C01852=1129.708,111.484,-56.807,-179.853,8.160,149.518
C01853=1129.704,111.733,-56.826,-179.851,8.164,149.518
C01854=1129.699,111.983,-56.846,-179.849,8.167,149.519
C01855=1129.694,112.232,-56.865,-179.847,8.171,149.519
C01856=1129.690,112.481,-56.884,-179.845,8.175,149.519
C01857=1129.684,112.730,-56.904,-179.843,8.178,149.520
C01858=1129.680,112.979,-56.923,-179.841,8.182,149.520
C01859=1129.674,113.228,-56.943,-179.839,8.185,149.520
C01860=1129.670,113.478,-56.962,-179.837,8.189,149.520
C01861=1129.665,113.727,-56.981,-179.835,8.193,149.521
C01862=1129.660,113.976,-57.001,-179.833,8.196,149.521
C01863=1129.655,114.226,-57.020,-179.831,8.200,149.521
C01864=1129.650,114.474,-57.040,-179.829,8.203,149.521
C01865=1129.646,114.724,-57.059,-179.828,8.207,149.522
C01866=1129.641,114.973,-57.078,-179.826,8.210,149.522
C01867=1129.636,115.222,-57.098,-179.823,8.214,149.522
C01868=1129.631,115.472,-57.117,-179.822,8.217,149.522
C01869=1129.627,115.721,-57.138,-179.820,8.220,149.523
C01870=1129.622,115.969,-57.156,-179.818,8.224,149.523
C01871=1129.618,116.184,-57.173,-179.816,8.228,149.523
C01872=1129.614,116.399,-57.190,-179.815,8.230,149.523
C01873=1129.610,116.614,-57.207,-179.813,8.233,149.524
C01874=1129.606,116.829,-57.224,-179.811,8.236,149.524
C01875=1129.601,117.043,-57.241,-179.810,8.239,149.524
C01876=1129.597,117.259,-57.258,-179.808,8.242,149.524
C01877=1129.593,117.474,-57.275,-179.806,8.245,149.525
C01878=1129.589,117.688,-57.292,-179.805,8.248,149.525
C01879=1129.584,117.938,-57.311,-179.803,8.252,149.525
C01880=1129.579,118.187,-57.331,-179.801,8.255,149.525
C01881=1129.574,118.435,-57.351,-179.799,8.259,149.525
C01882=1129.569,118.685,-57.371,-179.797,8.261,149.526
C01883=1129.565,118.935,-57.390,-179.796,8.265,149.526
C01884=1129.560,119.183,-57.409,-179.794,8.269,149.526
C01885=1129.556,119.432,-57.429,-179.792,8.272,149.527
C01886=1129.551,119.682,-57.449,-179.789,8.276,149.527
C01887=1129.546,119.931,-57.469,-179.787,8.279,149.527
C01888=1129.541,120.179,-57.489,-179.786,8.282,149.527
C01889=1129.536,120.429,-57.508,-179.784,8.286,149.528
C01890=1129.532,120.679,-57.528,-179.782,8.289,149.528
C01891=1129.527,120.928,-57.548,-179.780,8.293,149.528
C01892=1129.522,121.176,-57.568,-179.779,8.296,149.528
C01893=1129.517,121.425,-57.588,-179.777,8.299,149.528
C01894=1129.513,121.675,-57.608,-179.775,8.303,149.529
C01895=1129.508,121.925,-57.627,-179.773,8.306,149.529
C01896=1129.503,122.173,-57.647,-179.771,8.310,149.529
C01897=1129.498,122.422,-57.667,-179.770,8.313,149.530
C01898=1129.494,122.671,-57.687,-179.767,8.316,149.530
C01899=1129.489,122.921,-57.707,-179.766,8.320,149.530
C01900=1129.484,123.170,-57.728,-179.764,8.323,149.530
C01901=1129.478,123.419,-57.747,-179.762,8.326,149.531
C01902=1129.474,123.668,-57.768,-179.760,8.330,149.531
C01903=1129.469,123.918,-57.787,-179.759,8.334,149.531
C01904=1129.465,124.166,-57.808,-179.757,8.337,149.532
C01905=1129.460,124.416,-57.827,-179.755,8.340,149.532
C01906=1129.456,124.665,-57.848,-179.753,8.343,149.532
C01907=1129.450,124.914,-57.867,-179.751,8.347,149.532
C01908=1129.446,125.163,-57.887,-179.750,8.350,149.533
C01909=1129.441,125.412,-57.907,-179.748,8.353,149.533
C01910=1129.436,125.662,-57.928,-179.746,8.357,149.533
C01911=1129.431,125.911,-57.948,-179.744,8.360,149.533
C01912=1129.427,126.160,-57.968,-179.743,8.363,149.534
C01913=1129.422,126.409,-57.988,-179.741,8.367,149.534
C01914=1129.417,126.658,-58.008,-179.739,8.370,149.534
C01915=1129.413,126.907,-58.028,-179.737,8.373,149.534
C01916=1129.407,127.156,-58.049,-179.735,8.377,149.535
C01917=1129.403,127.406,-58.069,-179.733,8.381,149.535
C01918=1129.398,127.655,-58.089,-179.732,8.383,149.535
C01919=1129.394,127.904,-58.109,-179.730,8.387,149.536
C01920=1129.389,128.153,-58.129,-179.728,8.391,149.536
C01921=1129.384,128.402,-58.150,-179.727,8.393,149.536
C01922=1129.379,128.651,-58.170,-179.725,8.397,149.536
C01923=1129.374,128.900,-58.190,-179.723,8.400,149.537
C01924=1129.370,129.149,-58.210,-179.722,8.403,149.537
C01925=1129.364,129.398,-58.231,-179.720,8.407,149.537
C01926=1129.360,129.647,-58.251,-179.718,8.410,149.538
C01927=1129.356,129.863,-58.268,-179.717,8.412,149.538
C01928=1129.352,130.077,-58.286,-179.715,8.416,149.538
C01929=1129.348,130.292,-58.305,-179.713,8.419,149.538
C01930=1129.343,130.506,-58.321,-179.712,8.422,149.539
C01931=1129.340,130.721,-58.339,-179.711,8.424,149.539
C01932=1129.336,130.936,-58.356,-179.709,8.427,149.539
C01933=1129.331,131.151,-58.375,-179.708,8.430,149.539
C01934=1129.327,131.366,-58.392,-179.707,8.432,149.539
C01935=1129.323,131.615,-58.412,-179.704,8.436,149.540
C01936=1129.318,131.864,-58.433,-179.703,8.439,149.540
C01937=1129.313,132.113,-58.453,-179.701,8.443,149.540
C01938=1129.309,132.362,-58.474,-179.699,8.446,149.541
C01939=1129.304,132.611,-58.495,-179.698,8.449,149.541
C01940=1129.299,132.859,-58.515,-179.696,8.453,149.541
C01941=1129.294,133.108,-58.535,-179.695,8.455,149.541
C01942=1129.289,133.358,-58.556,-179.693,8.459,149.542
C01943=1129.284,133.607,-58.576,-179.692,8.462,149.542
C01944=1129.279,133.856,-58.597,-179.690,8.466,149.543
C01945=1129.275,134.105,-58.617,-179.688,8.469,149.543
C01946=1129.270,134.354,-58.637,-179.687,8.472,149.543
C01947=1129.266,134.604,-58.659,-179.685,8.476,149.543
C01948=1129.261,134.853,-58.679,-179.683,8.479,149.544
C01949=1129.256,135.103,-58.700,-179.681,8.482,149.544
C01950=1129.252,135.352,-58.720,-179.680,8.485,149.544
C01951=1129.247,135.600,-58.741,-179.678,8.489,149.545
C01952=1129.242,135.850,-58.762,-179.677,8.492,149.545
C01953=1129.238,136.099,-58.782,-179.675,8.495,149.545
C01954=1129.233,136.348,-58.803,-179.674,8.498,149.545
C01955=1129.228,136.597,-58.823,-179.672,8.502,149.546
C01956=1129.223,136.846,-58.844,-179.671,8.505,149.546
C01957=1129.219,137.094,-58.865,-179.669,8.508,149.547
C01958=1129.214,137.344,-58.886,-179.667,8.512,149.547
C01959=1129.209,137.593,-58.907,-179.666,8.515,149.547
C01960=1129.204,137.842,-58.928,-179.664,8.519,149.547
C01961=1129.200,138.091,-58.948,-179.663,8.522,149.548
C01962=1129.194,138.340,-58.969,-179.661,8.525,149.548
C01963=1129.190,138.589,-58.990,-179.660,8.528,149.549
C01964=1129.185,138.838,-59.010,-179.658,8.532,149.549
C01965=1129.181,139.087,-59.032,-179.657,8.535,149.549
C01966=1129.176,139.337,-59.053,-179.655,8.537,149.549
C01967=1129.172,139.586,-59.073,-179.654,8.541,149.550
C01968=1129.166,139.835,-59.094,-179.652,8.544,149.550
C01969=1129.162,140.084,-59.115,-179.651,8.548,149.550
C01970=1129.157,140.333,-59.136,-179.649,8.551,149.551
C01971=1129.152,140.582,-59.157,-179.647,8.555,149.551
C01972=1129.148,140.831,-59.178,-179.646,8.557,149.551
C01973=1129.143,141.081,-59.199,-179.644,8.561,149.552
C01974=1129.139,141.330,-59.219,-179.643,8.564,149.552
C01975=1129.134,141.578,-59.241,-179.641,8.568,149.552
C01976=1129.129,141.827,-59.261,-179.640,8.571,149.553
C01977=1129.124,142.076,-59.282,-179.638,8.574,149.553
C01978=1129.119,142.326,-59.303,-179.637,8.577,149.554
C01979=1129.115,142.574,-59.324,-179.635,8.581,149.554
C01980=1129.110,142.824,-59.346,-179.634,8.584,149.554
C01981=1129.105,143.073,-59.367,-179.633,8.587,149.555
C01982=1129.101,143.322,-59.388,-179.631,8.590,149.555
C01983=1129.096,143.536,-59.406,-179.630,8.594,149.555
C01984=1129.093,143.751,-59.424,-179.629,8.596,149.556
C01985=1129.088,143.966,-59.442,-179.627,8.599,149.556
C01986=1129.085,144.180,-59.460,-179.626,8.602,149.556
C01987=1129.080,144.395,-59.478,-179.625,8.605,149.556
C01988=1129.076,144.610,-59.497,-179.624,8.608,149.557
C01989=1129.072,144.824,-59.515,-179.622,8.611,149.557
C01990=1129.068,145.039,-59.533,-179.622,8.613,149.557
C01991=1129.063,145.288,-59.555,-179.619,8.617,149.558
C01992=1129.059,145.537,-59.575,-179.616,8.621,149.558
C01993=1129.054,145.786,-59.597,-179.613,8.625,149.558
C01994=1129.049,146.035,-59.618,-179.611,8.630,149.558
C01995=1129.045,146.284,-59.639,-179.607,8.633,149.558
C01996=1129.040,146.533,-59.660,-179.605,8.637,149.558
C01997=1129.036,146.782,-59.682,-179.603,8.641,149.559
C01998=1129.030,147.031,-59.703,-179.600,8.646,149.559
C01999=1129.026,147.280,-59.725,-179.597,8.649,149.559
C02000=1129.021,147.529,-59.745,-179.595,8.653,149.559
C02001=1129.017,147.778,-59.767,-179.592,8.657,149.559
C02002=1129.012,148.028,-59.788,-179.589,8.661,149.559
C02003=1129.007,148.276,-59.810,-179.587,8.665,149.560
C02004=1129.002,148.525,-59.832,-179.584,8.669,149.560
C02005=1128.998,148.775,-59.852,-179.581,8.673,149.560
C02006=1128.993,149.023,-59.874,-179.579,8.676,149.560
C02007=1128.988,149.272,-59.895,-179.576,8.680,149.560
C02008=1128.984,149.522,-59.917,-179.573,8.684,149.560
C02009=1128.979,149.770,-59.939,-179.571,8.688,149.561
C02010=1128.974,150.020,-59.960,-179.568,8.692,149.561
C02011=1128.969,150.269,-59.982,-179.565,8.696,149.561
C02012=1128.965,150.518,-60.003,-179.562,8.699,149.561
C02013=1128.960,150.766,-60.025,-179.560,8.703,149.561
C02014=1128.955,151.016,-60.046,-179.557,8.706,149.561
C02015=1128.951,151.265,-60.067,-179.554,8.711,149.561
C02016=1128.946,151.513,-60.089,-179.552,8.714,149.561
C02017=1128.942,151.763,-60.111,-179.549,8.718,149.562
C02018=1128.937,152.011,-60.133,-179.547,8.721,149.562
C02019=1128.932,152.261,-60.154,-179.544,8.725,149.562
C02020=1128.928,152.510,-60.176,-179.541,8.729,149.562
C02021=1128.923,152.759,-60.198,-179.539,8.733,149.562
C02022=1128.918,153.008,-60.220,-179.536,8.736,149.562
C02023=1128.914,153.256,-60.241,-179.534,8.740,149.563
C02024=1128.909,153.505,-60.263,-179.531,8.743,149.563
C02025=1128.904,153.754,-60.285,-179.528,8.748,149.563
C02026=1128.899,154.004,-60.306,-179.526,8.751,149.563
C02027=1128.894,154.253,-60.329,-179.523,8.755,149.563
C02028=1128.889,154.502,-60.350,-179.521,8.758,149.563
C02029=1128.885,154.751,-60.372,-179.518,8.761,149.563
C02030=1128.880,155.000,-60.394,-179.515,8.765,149.563
C02031=1128.876,155.249,-60.416,-179.513,8.768,149.563
C02032=1128.871,155.498,-60.438,-179.510,8.773,149.564
C02033=1128.866,155.747,-60.459,-179.508,8.776,149.564
C02034=1128.862,155.996,-60.482,-179.505,8.779,149.564
C02035=1128.857,156.245,-60.503,-179.502,8.783,149.564
C02036=1128.853,156.494,-60.525,-179.500,8.786,149.564
C02037=1128.847,156.743,-60.548,-179.498,8.790,149.564
C02038=1128.843,156.992,-60.570,-179.495,8.794,149.564
C02039=1128.839,157.206,-60.589,-179.493,8.796,149.564
C02040=1128.835,157.421,-60.608,-179.491,8.800,149.564
C02041=1128.831,157.636,-60.627,-179.488,8.803,149.564
C02042=1128.827,157.850,-60.646,-179.486,8.805,149.564
C02043=1128.823,158.065,-60.665,-179.484,8.808,149.565
C02044=1128.819,158.279,-60.684,-179.482,8.812,149.565
C02045=1128.815,158.494,-60.703,-179.480,8.814,149.565
C02046=1128.811,158.708,-60.722,-179.477,8.817,149.565
C02047=1128.806,158.956,-60.744,-179.475,8.820,149.565
C02048=1128.802,159.206,-60.766,-179.473,8.824,149.565
C02049=1128.797,159.455,-60.789,-179.469,8.827,149.565
C02050=1128.793,159.703,-60.811,-179.467,8.831,149.565
C02051=1128.788,159.953,-60.833,-179.465,8.834,149.565
C02052=1128.783,160.201,-60.855,-179.462,8.837,149.565
C02053=1128.778,160.451,-60.877,-179.460,8.841,149.566
C02054=1128.774,160.699,-60.900,-179.457,8.845,149.566
C02055=1128.770,160.948,-60.922,-179.454,8.848,149.566
C02056=1128.765,161.198,-60.944,-179.452,8.851,149.566
C02057=1128.760,161.446,-60.967,-179.450,8.854,149.566
C02058=1128.756,161.695,-60.989,-179.447,8.857,149.566
C02059=1128.751,161.944,-61.011,-179.445,8.860,149.566
C02060=1128.746,162.193,-61.034,-179.443,8.864,149.566
C02061=1128.742,162.442,-61.056,-179.440,8.868,149.566
C02062=1128.737,162.690,-61.078,-179.437,8.871,149.566
C02063=1128.732,162.940,-61.101,-179.435,8.874,149.566
C02064=1128.728,163.189,-61.123,-179.432,8.878,149.567
C02065=1128.723,163.438,-61.146,-179.430,8.881,149.567
C02066=1128.718,163.687,-61.168,-179.427,8.884,149.567
C02067=1128.714,163.936,-61.191,-179.425,8.887,149.567
C02068=1128.709,164.185,-61.213,-179.423,8.890,149.567
C02069=1128.705,164.434,-61.236,-179.420,8.893,149.567
C02070=1128.700,164.683,-61.259,-179.418,8.897,149.567
C02071=1128.695,164.931,-61.281,-179.415,8.900,149.567
C02072=1128.691,165.181,-61.303,-179.413,8.903,149.567
C02073=1128.686,165.430,-61.326,-179.411,8.906,149.567
C02074=1128.682,165.678,-61.348,-179.408,8.909,149.567
C02075=1128.677,165.927,-61.371,-179.406,8.912,149.567
C02076=1128.673,166.177,-61.394,-179.403,8.916,149.568
C02077=1128.668,166.426,-61.417,-179.401,8.919,149.568
C02078=1128.663,166.674,-61.439,-179.398,8.922,149.568
C02079=1128.658,166.923,-61.462,-179.396,8.925,149.568
C02080=1128.654,167.172,-61.485,-179.394,8.929,149.568
C02081=1128.649,167.421,-61.507,-179.391,8.932,149.568
C02082=1128.645,167.670,-61.530,-179.389,8.935,149.568
C02083=1128.640,167.919,-61.553,-179.387,8.937,149.568
C02084=1128.636,168.168,-61.575,-179.385,8.941,149.568
C02085=1128.630,168.416,-61.598,-179.382,8.944,149.568
C02086=1128.626,168.665,-61.622,-179.380,8.947,149.568
C02087=1128.622,168.915,-61.644,-179.377,8.950,149.568
C02088=1128.617,169.164,-61.667,-179.375,8.954,149.569
C02089=1128.612,169.412,-61.689,-179.373,8.957,149.569
C02090=1128.608,169.661,-61.713,-179.370,8.960,149.569
C02091=1128.603,169.911,-61.735,-179.368,8.962,149.569
C02092=1128.599,170.159,-61.758,-179.366,8.966,149.569
C02093=1128.594,170.408,-61.781,-179.364,8.969,149.569
C02094=1128.589,170.656,-61.804,-179.361,8.972,149.569
C02095=1128.585,170.872,-61.824,-179.359,8.974,149.569
C02096=1128.581,171.085,-61.844,-179.357,8.978,149.569
C02097=1128.577,171.300,-61.864,-179.355,8.980,149.569
C02098=1128.573,171.514,-61.883,-179.353,8.982,149.569
C02099=1128.570,171.729,-61.903,-179.351,8.985,149.569
C02100=1128.565,171.943,-61.923,-179.349,8.988,149.570
C02101=1128.562,172.158,-61.943,-179.347,8.990,149.570
C02102=1128.557,172.372,-61.963,-179.345,8.993,149.570
C02103=1128.553,172.621,-61.985,-179.343,8.996,149.570
C02104=1128.548,172.870,-62.009,-179.341,8.999,149.570
C02105=1128.544,173.119,-62.032,-179.339,9.002,149.570
C02106=1128.540,173.368,-62.055,-179.336,9.005,149.570
C02107=1128.535,173.617,-62.078,-179.334,9.008,149.570
C02108=1128.530,173.865,-62.101,-179.332,9.011,149.570
C02109=1128.525,174.114,-62.124,-179.330,9.014,149.570
C02110=1128.521,174.363,-62.147,-179.327,9.017,149.570
C02111=1128.516,174.612,-62.171,-179.325,9.020,149.570
C02112=1128.512,174.861,-62.194,-179.323,9.023,149.571
C02113=1128.507,175.110,-62.217,-179.321,9.026,149.571
C02114=1128.503,175.358,-62.240,-179.318,9.029,149.571
C02115=1128.498,175.607,-62.263,-179.317,9.032,149.571
C02116=1128.494,175.857,-62.287,-179.314,9.035,149.571
C02117=1128.488,176.105,-62.310,-179.312,9.038,149.571
C02118=1128.484,176.354,-62.333,-179.310,9.040,149.571
C02119=1128.480,176.603,-62.356,-179.308,9.044,149.571
C02120=1128.475,176.852,-62.379,-179.305,9.047,149.571
C02121=1128.470,177.101,-62.403,-179.304,9.049,149.572
C02122=1128.465,177.350,-62.426,-179.301,9.053,149.572
C02123=1128.461,177.599,-62.449,-179.299,9.056,149.572
C02124=1128.456,177.848,-62.473,-179.297,9.058,149.572
C02125=1128.452,178.096,-62.496,-179.295,9.061,149.572
C02126=1128.448,178.345,-62.520,-179.293,9.064,149.572
C02127=1128.443,178.594,-62.543,-179.291,9.067,149.572
C02128=1128.438,178.843,-62.566,-179.288,9.070,149.572
C02129=1128.434,179.092,-62.590,-179.287,9.073,149.572
C02130=1128.429,179.340,-62.614,-179.284,9.076,149.572
C02131=1128.425,179.589,-62.637,-179.281,9.080,149.572
C02132=1128.420,179.838,-62.660,-179.278,9.084,149.572
C02133=1128.415,180.088,-62.684,-179.275,9.087,149.572
C02134=1128.411,180.336,-62.707,-179.272,9.090,149.572
C02135=1128.407,180.585,-62.731,-179.269,9.093,149.572
C02136=1128.402,180.834,-62.754,-179.266,9.097,149.572
C02137=1128.397,181.083,-62.777,-179.263,9.100,149.572
C02138=1128.393,181.331,-62.801,-179.260,9.104,149.572
C02139=1128.388,181.580,-62.825,-179.257,9.107,149.572
C02140=1128.384,181.829,-62.848,-179.254,9.110,149.572
C02141=1128.379,182.078,-62.872,-179.251,9.114,149.572
C02142=1128.375,182.327,-62.896,-179.249,9.117,149.572
C02143=1128.370,182.575,-62.920,-179.246,9.119,149.572
C02144=1128.365,182.824,-62.943,-179.243,9.122,149.572
C02145=1128.361,183.073,-62.966,-179.240,9.126,149.572
C02146=1128.356,183.322,-62.990,-179.237,9.129,149.572
C02147=1128.351,183.571,-63.014,-179.234,9.132,149.572
C02148=1128.347,183.820,-63.039,-179.232,9.135,149.572
C02149=1128.342,184.069,-63.062,-179.229,9.138,149.572
C02150=1128.338,184.317,-63.086,-179.227,9.142,149.572
C02151=1128.333,184.531,-63.107,-179.224,9.144,149.572
C02152=1128.330,184.746,-63.127,-179.222,9.147,149.572
C02153=1128.326,184.960,-63.148,-179.219,9.150,149.572
C02154=1128.322,185.175,-63.168,-179.218,9.152,149.572
C02155=1128.318,185.389,-63.189,-179.216,9.154,149.572
C02156=1128.315,185.603,-63.209,-179.213,9.157,149.572
C02157=1128.311,185.817,-63.230,-179.211,9.159,149.572
C02158=1128.306,186.031,-63.250,-179.209,9.162,149.572
C02159=1128.303,186.280,-63.275,-179.206,9.165,149.572
C02160=1128.298,186.530,-63.298,-179.204,9.168,149.572
C02161=1128.293,186.778,-63.323,-179.201,9.171,149.572
C02162=1128.288,187.027,-63.347,-179.199,9.174,149.572
C02163=1128.284,187.276,-63.370,-179.197,9.176,149.572
C02164=1128.279,187.524,-63.394,-179.194,9.180,149.572
C02165=1128.275,187.772,-63.418,-179.192,9.183,149.572
C02166=1128.270,188.023,-63.442,-179.190,9.185,149.572
C02167=1128.266,188.271,-63.467,-179.187,9.188,149.572
C02168=1128.261,188.519,-63.491,-179.185,9.191,149.572
C02169=1128.257,188.768,-63.514,-179.183,9.194,149.572
C02170=1128.251,189.017,-63.539,-179.181,9.197,149.573
C02171=1128.248,189.266,-63.563,-179.179,9.199,149.573
C02172=1128.243,189.515,-63.587,-179.176,9.202,149.573
C02173=1128.238,189.764,-63.610,-179.174,9.204,149.573
C02174=1128.233,190.012,-63.635,-179.172,9.208,149.573
C02175=1128.229,190.261,-63.659,-179.170,9.210,149.573
C02176=1128.225,190.510,-63.684,-179.168,9.212,149.573
C02177=1128.220,190.759,-63.708,-179.165,9.215,149.573
C02178=1128.215,191.008,-63.732,-179.163,9.218,149.573
C02179=1128.211,191.256,-63.756,-179.161,9.221,149.573
C02180=1128.207,191.505,-63.780,-179.160,9.223,149.573
C02181=1128.202,191.754,-63.805,-179.158,9.226,149.573
C02182=1128.198,192.002,-63.829,-179.156,9.228,149.573
C02183=1128.192,192.251,-63.854,-179.154,9.232,149.573
C02184=1128.189,192.500,-63.878,-179.152,9.234,149.573
C02185=1128.184,192.749,-63.901,-179.150,9.236,149.573
C02186=1128.179,192.998,-63.926,-179.148,9.239,149.574
C02187=1128.174,193.246,-63.950,-179.146,9.241,149.574
C02188=1128.171,193.495,-63.975,-179.145,9.244,149.574
C02189=1128.166,193.744,-63.999,-179.143,9.246,149.574
C02190=1128.161,193.993,-64.023,-179.141,9.250,149.574
C02191=1128.157,194.241,-64.047,-179.139,9.252,149.574
C02192=1128.152,194.490,-64.072,-179.138,9.255,149.575
C02193=1128.148,194.739,-64.097,-179.136,9.257,149.575
C02194=1128.143,194.988,-64.121,-179.134,9.260,149.575
C02195=1128.139,195.237,-64.146,-179.133,9.263,149.575
C02196=1128.134,195.485,-64.170,-179.132,9.264,149.575
C02197=1128.129,195.734,-64.194,-179.130,9.267,149.575
C02198=1128.126,195.983,-64.219,-179.129,9.270,149.576
C02199=1128.120,196.232,-64.244,-179.127,9.272,149.576
C02200=1128.116,196.480,-64.268,-179.124,9.276,149.576
C02201=1128.112,196.730,-64.293,-179.119,9.280,149.576
C02202=1128.107,196.978,-64.317,-179.116,9.284,149.575
C02203=1128.102,197.227,-64.341,-179.112,9.287,149.575
C02204=1128.098,197.476,-64.366,-179.108,9.291,149.575
C02205=1128.093,197.724,-64.390,-179.104,9.295,149.575
C02206=1128.089,197.972,-64.415,-179.101,9.298,149.575
C02207=1128.085,198.187,-64.436,-179.097,9.302,149.575
C02208=1128.081,198.401,-64.458,-179.094,9.305,149.575
C02209=1128.077,198.616,-64.479,-179.091,9.308,149.574
C02210=1128.073,198.830,-64.500,-179.088,9.311,149.574
C02211=1128.070,199.044,-64.522,-179.085,9.314,149.574
C02212=1128.066,199.258,-64.543,-179.081,9.317,149.574
C02213=1128.062,199.472,-64.564,-179.079,9.320,149.574
C02214=1128.058,199.686,-64.586,-179.076,9.323,149.574
C02215=1128.053,199.935,-64.610,-179.072,9.327,149.574
C02216=1128.049,200.184,-64.635,-179.069,9.330,149.574
C02217=1128.045,200.432,-64.660,-179.065,9.334,149.573
C02218=1128.040,200.681,-64.685,-179.062,9.336,149.573
C02219=1128.035,200.930,-64.710,-179.058,9.340,149.573
C02220=1128.031,201.178,-64.735,-179.055,9.343,149.573
C02221=1128.026,201.427,-64.760,-179.052,9.346,149.573
C02222=1128.021,201.676,-64.784,-179.048,9.350,149.573
C02223=1128.018,201.925,-64.809,-179.045,9.352,149.573
C02224=1128.013,202.173,-64.834,-179.042,9.356,149.572
C02225=1128.008,202.422,-64.860,-179.039,9.359,149.572
C02226=1128.004,202.671,-64.884,-179.035,9.362,149.572
C02227=1128.000,202.919,-64.910,-179.032,9.365,149.572
C02228=1127.995,203.168,-64.934,-179.029,9.368,149.572
C02229=1127.990,203.417,-64.960,-179.026,9.371,149.572
C02230=1127.986,203.665,-64.984,-179.023,9.374,149.572
C02231=1127.982,203.914,-65.010,-179.020,9.377,149.571
C02232=1127.977,204.163,-65.035,-179.017,9.380,149.572
C02233=1127.973,204.412,-65.060,-179.014,9.383,149.571
C02234=1127.969,204.661,-65.085,-179.011,9.386,149.571
C02235=1127.964,204.909,-65.110,-179.008,9.389,149.571
C02236=1127.960,205.158,-65.136,-179.005,9.392,149.571
C02237=1127.955,205.406,-65.161,-179.002,9.394,149.571
C02238=1127.950,205.655,-65.186,-178.999,9.397,149.571
C02239=1127.945,205.904,-65.211,-178.996,9.400,149.571
C02240=1127.941,206.153,-65.237,-178.994,9.403,149.571
C02241=1127.937,206.401,-65.262,-178.991,9.406,149.571
C02242=1127.932,206.650,-65.287,-178.988,9.409,149.571
C02243=1127.928,206.899,-65.312,-178.986,9.411,149.570
C02244=1127.923,207.147,-65.338,-178.984,9.414,149.571
C02245=1127.919,207.396,-65.363,-178.981,9.417,149.570
C02246=1127.915,207.645,-65.388,-178.978,9.420,149.570
C02247=1127.910,207.893,-65.414,-178.976,9.422,149.570
C02248=1127.905,208.142,-65.440,-178.973,9.425,149.570
C02249=1127.901,208.390,-65.465,-178.970,9.428,149.570
C02250=1127.896,208.640,-65.490,-178.968,9.430,149.570
C02251=1127.892,208.888,-65.516,-178.966,9.433,149.570
C02252=1127.887,209.136,-65.541,-178.964,9.435,149.570
C02253=1127.884,209.385,-65.566,-178.961,9.438,149.570
C02254=1127.879,209.634,-65.592,-178.959,9.441,149.570
C02255=1127.874,209.882,-65.617,-178.957,9.444,149.570
C02256=1127.870,210.131,-65.642,-178.955,9.446,149.570
C02257=1127.866,210.380,-65.668,-178.953,9.448,149.570
C02258=1127.861,210.628,-65.694,-178.950,9.451,149.570
C02259=1127.857,210.877,-65.719,-178.948,9.454,149.570
C02260=1127.853,211.126,-65.745,-178.947,9.456,149.571
C02261=1127.848,211.374,-65.771,-178.944,9.459,149.571
C02262=1127.843,211.623,-65.796,-178.943,9.462,149.571
C02263=1127.839,211.837,-65.818,-178.941,9.464,149.571
C02264=1127.835,212.051,-65.840,-178.939,9.466,149.571
C02265=1127.831,212.265,-65.862,-178.937,9.468,149.571
C02266=1127.828,212.480,-65.885,-178.936,9.471,149.571
C02267=1127.824,212.694,-65.907,-178.935,9.472,149.571
C02268=1127.820,212.908,-65.929,-178.933,9.475,149.571
C02269=1127.816,213.121,-65.951,-178.931,9.477,149.572
C02270=1127.812,213.335,-65.973,-178.931,9.479,149.572
C02271=1127.808,213.584,-65.999,-178.929,9.482,149.572
C02272=1127.804,213.833,-66.024,-178.927,9.485,149.572
C02273=1127.799,214.081,-66.050,-178.925,9.487,149.572
C02274=1127.795,214.330,-66.076,-178.923,9.490,149.572
C02275=1127.790,214.579,-66.101,-178.921,9.492,149.572
C02276=1127.786,214.828,-66.127,-178.919,9.496,149.572
C02277=1127.781,215.076,-66.153,-178.917,9.498,149.573
C02278=1127.776,215.325,-66.179,-178.915,9.501,149.573
C02279=1127.772,215.574,-66.204,-178.913,9.504,149.573
C02280=1127.768,215.822,-66.230,-178.911,9.506,149.573
C02281=1127.763,216.070,-66.256,-178.909,9.510,149.573
C02282=1127.759,216.319,-66.282,-178.907,9.512,149.573
C02283=1127.755,216.567,-66.308,-178.905,9.515,149.573
C02284=1127.751,216.816,-66.334,-178.903,9.519,149.574
C02285=1127.745,217.065,-66.360,-178.901,9.521,149.574
C02286=1127.741,217.313,-66.385,-178.898,9.524,149.574
C02287=1127.737,217.562,-66.411,-178.896,9.528,149.574
C02288=1127.733,217.810,-66.438,-178.894,9.530,149.574
C02289=1127.729,218.059,-66.463,-178.892,9.533,149.574
C02290=1127.723,218.308,-66.489,-178.889,9.536,149.574
C02291=1127.719,218.556,-66.515,-178.887,9.540,149.574
C02292=1127.715,218.805,-66.541,-178.885,9.542,149.575
C02293=1127.711,219.053,-66.567,-178.883,9.545,149.575
C02294=1127.706,219.303,-66.594,-178.880,9.548,149.575
C02295=1127.701,219.551,-66.619,-178.878,9.551,149.575
C02296=1127.697,219.800,-66.645,-178.875,9.554,149.575
C02297=1127.693,220.048,-66.671,-178.873,9.558,149.575
C02298=1127.688,220.297,-66.698,-178.871,9.561,149.575
C02299=1127.684,220.546,-66.723,-178.868,9.564,149.575
C02300=1127.680,220.794,-66.750,-178.865,9.567,149.575
C02301=1127.675,221.043,-66.776,-178.863,9.570,149.575
C02302=1127.670,221.292,-66.802,-178.860,9.573,149.575
C02303=1127.666,221.539,-66.828,-178.858,9.577,149.575
C02304=1127.662,221.788,-66.854,-178.855,9.580,149.575
C02305=1127.657,222.036,-66.881,-178.852,9.584,149.576
C02306=1127.653,222.285,-66.907,-178.849,9.586,149.575
C02307=1127.648,222.534,-66.933,-178.847,9.589,149.575
C02308=1127.644,222.783,-66.959,-178.844,9.593,149.576
C02309=1127.640,223.031,-66.985,-178.841,9.596,149.576
C02310=1127.635,223.280,-67.012,-178.838,9.600,149.576
C02311=1127.631,223.529,-67.038,-178.835,9.603,149.576
C02312=1127.626,223.777,-67.065,-178.832,9.606,149.576
C02313=1127.621,224.025,-67.090,-178.830,9.609,149.576
C02314=1127.617,224.273,-67.117,-178.826,9.613,149.576
C02315=1127.612,224.523,-67.143,-178.824,9.616,149.576
C02316=1127.609,224.771,-67.170,-178.821,9.620,149.576
C02317=1127.604,225.020,-67.196,-178.818,9.623,149.576
C02318=1127.600,225.268,-67.222,-178.814,9.626,149.576
C02319=1127.596,225.482,-67.246,-178.812,9.629,149.576
C02320=1127.592,225.696,-67.268,-178.809,9.632,149.576
C02321=1127.588,225.910,-67.291,-178.806,9.635,149.575
C02322=1127.585,226.124,-67.314,-178.804,9.638,149.576
C02323=1127.581,226.338,-67.337,-178.801,9.641,149.575
C02324=1127.577,226.551,-67.360,-178.798,9.644,149.575
C02325=1127.573,226.766,-67.382,-178.795,9.647,149.575
C02326=1127.569,226.980,-67.405,-178.792,9.649,149.575
C02327=1127.565,227.228,-67.432,-178.790,9.653,149.575
C02328=1127.560,227.477,-67.459,-178.786,9.656,149.575
C02329=1127.556,227.725,-67.485,-178.782,9.660,149.575
C02330=1127.551,227.974,-67.511,-178.779,9.663,149.575
C02331=1127.547,228.222,-67.538,-178.775,9.667,149.575
C02332=1127.543,228.471,-67.565,-178.772,9.669,149.575
C02333=1127.538,228.719,-67.592,-178.769,9.673,149.575
C02334=1127.534,228.967,-67.619,-178.765,9.676,149.574
C02335=1127.529,229.216,-67.645,-178.762,9.680,149.574
C02336=1127.526,229.465,-67.672,-178.758,9.683,149.574
C02337=1127.521,229.714,-67.699,-178.754,9.687,149.574
C02338=1127.517,229.962,-67.726,-178.751,9.691,149.574
C02339=1127.513,230.211,-67.752,-178.747,9.694,149.574
C02340=1127.508,230.459,-67.779,-178.743,9.697,149.574
C02341=1127.503,230.708,-67.806,-178.740,9.701,149.573
C02342=1127.499,230.956,-67.833,-178.737,9.703,149.573
C02343=1127.495,231.204,-67.860,-178.733,9.707,149.573
C02344=1127.490,231.453,-67.887,-178.730,9.711,149.573
C02345=1127.486,231.702,-67.914,-178.726,9.713,149.573
C02346=1127.481,231.950,-67.941,-178.723,9.716,149.573
C02347=1127.478,232.199,-67.968,-178.719,9.720,149.573
C02348=1127.473,232.447,-67.995,-178.716,9.723,149.572
C02349=1127.468,232.696,-68.022,-178.713,9.725,149.572
C02350=1127.464,232.944,-68.049,-178.710,9.729,149.572
C02351=1127.460,233.192,-68.076,-178.707,9.732,149.572
C02352=1127.456,233.441,-68.103,-178.703,9.735,149.572
C02353=1127.451,233.690,-68.130,-178.700,9.738,149.572
C02354=1127.447,233.938,-68.158,-178.697,9.740,149.571
C02355=1127.442,234.186,-68.185,-178.694,9.743,149.571
C02356=1127.437,234.435,-68.212,-178.690,9.747,149.571
C02357=1127.434,234.684,-68.239,-178.687,9.749,149.571
C02358=1127.429,234.932,-68.266,-178.684,9.752,149.571
C02359=1127.425,235.180,-68.294,-178.681,9.755,149.571
C02360=1127.420,235.429,-68.321,-178.678,9.758,149.571
C02361=1127.416,235.678,-68.348,-178.675,9.760,149.571
C02362=1127.412,235.926,-68.375,-178.673,9.763,149.571
C02363=1127.407,236.174,-68.403,-178.670,9.766,149.571
C02364=1127.403,236.423,-68.430,-178.667,9.769,149.570
C02365=1127.398,236.672,-68.457,-178.665,9.771,149.570
C02366=1127.395,236.920,-68.484,-178.662,9.774,149.570
C02367=1127.390,237.168,-68.512,-178.659,9.776,149.570
C02368=1127.386,237.416,-68.539,-178.656,9.779,149.570
C02369=1127.382,237.666,-68.566,-178.654,9.782,149.570
C02370=1127.377,237.913,-68.594,-178.651,9.784,149.570
C02371=1127.372,238.162,-68.621,-178.648,9.787,149.570
C02372=1127.368,238.410,-68.649,-178.646,9.789,149.570
C02373=1127.364,238.659,-68.676,-178.643,9.792,149.570
C02374=1127.359,238.908,-68.703,-178.641,9.794,149.569
C02375=1127.356,239.122,-68.728,-178.639,9.796,149.569
C02376=1127.352,239.335,-68.751,-178.637,9.798,149.569
C02377=1127.348,239.549,-68.774,-178.634,9.800,149.569
C02378=1127.344,239.762,-68.799,-178.633,9.803,149.569
C02379=1127.341,239.976,-68.822,-178.630,9.805,149.569
C02380=1127.337,240.190,-68.846,-178.628,9.807,149.569
C02381=1127.333,240.404,-68.870,-178.626,9.809,149.569
C02382=1127.330,240.617,-68.894,-178.624,9.811,149.569
C02383=1127.325,240.866,-68.921,-178.622,9.814,149.569
C02384=1127.321,241.115,-68.949,-178.620,9.816,149.569
C02385=1127.317,241.363,-68.976,-178.618,9.818,149.569
C02386=1127.312,241.611,-69.004,-178.615,9.821,149.569
C02387=1127.308,241.860,-69.032,-178.613,9.823,149.569
C02388=1127.303,242.108,-69.059,-178.611,9.825,149.569
C02389=1127.299,242.357,-69.086,-178.609,9.828,149.569
C02390=1127.295,242.605,-69.115,-178.607,9.830,149.569
C02391=1127.290,242.854,-69.142,-178.606,9.832,149.569
C02392=1127.286,243.102,-69.170,-178.603,9.834,149.569
C02393=1127.282,243.350,-69.198,-178.601,9.837,149.569
C02394=1127.277,243.599,-69.225,-178.599,9.839,149.569
C02395=1127.274,243.847,-69.253,-178.598,9.841,149.569
C02396=1127.269,244.096,-69.281,-178.596,9.843,149.569
C02397=1127.264,244.344,-69.308,-178.595,9.846,149.570
C02398=1127.260,244.593,-69.336,-178.593,9.848,149.570
C02399=1127.256,244.841,-69.364,-178.591,9.850,149.570
C02400=1127.252,245.090,-69.392,-178.589,9.853,149.570
C02401=1127.247,245.338,-69.419,-178.588,9.854,149.570
C02402=1127.242,245.586,-69.448,-178.586,9.857,149.570
C02403=1127.238,245.835,-69.475,-178.585,9.859,149.570
C02404=1127.234,246.083,-69.503,-178.584,9.861,149.570
C02405=1127.230,246.331,-69.531,-178.582,9.863,149.570
C02406=1127.225,246.580,-69.558,-178.581,9.865,149.570
C02407=1127.221,246.829,-69.587,-178.579,9.868,149.571
C02408=1127.217,247.077,-69.615,-178.578,9.870,149.571
C02409=1127.212,247.325,-69.642,-178.576,9.872,149.571
C02410=1127.208,247.574,-69.670,-178.572,9.876,149.571
C02411=1127.203,247.822,-69.698,-178.565,9.881,149.570
C02412=1127.199,248.071,-69.726,-178.559,9.886,149.570
C02413=1127.195,248.318,-69.754,-178.553,9.891,149.569
C02414=1127.191,248.567,-69.782,-178.546,9.896,149.569
C02415=1127.186,248.815,-69.811,-178.540,9.900,149.568
C02416=1127.182,249.064,-69.839,-178.535,9.905,149.568
C02417=1127.178,249.312,-69.867,-178.529,9.909,149.568
C02418=1127.173,249.561,-69.895,-178.524,9.914,149.567
C02419=1127.169,249.809,-69.922,-178.519,9.917,149.567
C02420=1127.165,250.057,-69.952,-178.514,9.921,149.566
C02421=1127.160,250.305,-69.980,-178.509,9.925,149.566
C02422=1127.157,250.554,-70.008,-178.505,9.928,149.566
C02423=1127.152,250.802,-70.036,-178.500,9.932,149.565
C02424=1127.148,251.050,-70.064,-178.496,9.935,149.565
C02425=1127.143,251.299,-70.093,-178.493,9.938,149.565
C02426=1127.139,251.547,-70.121,-178.489,9.941,149.565
C02427=1127.134,251.796,-70.149,-178.486,9.943,149.564
C02428=1127.130,252.044,-70.177,-178.483,9.946,149.564
C02429=1127.126,252.292,-70.207,-178.480,9.949,149.564
C02430=1127.122,252.541,-70.235,-178.478,9.951,149.564
C02431=1127.118,252.754,-70.259,-178.475,9.953,149.564
C02432=1127.114,252.968,-70.283,-178.473,9.955,149.564
C02433=1127.111,253.181,-70.308,-178.471,9.956,149.563
C02434=1127.107,253.395,-70.332,-178.470,9.957,149.563
C02435=1127.103,253.609,-70.357,-178.469,9.959,149.564
C02436=1127.100,253.823,-70.382,-178.467,9.961,149.564
C02437=1127.097,254.037,-70.406,-178.466,9.962,149.564
C02438=1127.092,254.250,-70.430,-178.465,9.964,149.564
C02439=1127.088,254.498,-70.460,-178.464,9.964,149.564
C02440=1127.084,254.747,-70.488,-178.463,9.966,149.564
C02441=1127.079,254.995,-70.516,-178.463,9.967,149.564
C02442=1127.075,255.244,-70.544,-178.463,9.969,149.564
C02443=1127.071,255.492,-70.574,-178.463,9.969,149.565
C02444=1127.066,255.740,-70.602,-178.463,9.970,149.565
C02445=1127.062,255.989,-70.630,-178.463,9.972,149.565
C02446=1127.058,256.237,-70.659,-178.460,9.974,149.565
C02447=1127.054,256.485,-70.687,-178.458,9.977,149.565
C02448=1127.049,256.734,-70.716,-178.455,9.980,149.565
C02449=1127.046,256.982,-70.744,-178.452,9.983,149.565
C02450=1127.041,257.230,-70.773,-178.449,9.986,149.565
C02451=1127.036,257.479,-70.802,-178.446,9.988,149.565
C02452=1127.033,257.727,-70.830,-178.443,9.991,149.565
C02453=1127.028,257.975,-70.859,-178.440,9.994,149.564
C02454=1127.024,258.223,-70.887,-178.437,9.997,149.564
C02455=1127.020,258.472,-70.917,-178.434,10.000,149.564
C02456=1127.015,258.720,-70.945,-178.431,10.003,149.564
C02457=1127.011,258.968,-70.973,-178.428,10.006,149.564
C02458=1127.007,259.217,-71.003,-178.424,10.009,149.564
C02459=1127.002,259.465,-71.031,-178.421,10.012,149.564
C02460=1126.998,259.713,-71.060,-178.418,10.014,149.564
C02461=1126.994,259.962,-71.089,-178.414,10.018,149.563
C02462=1126.990,260.210,-71.118,-178.411,10.021,149.563
C02463=1126.985,260.458,-71.147,-178.409,10.024,149.563
C02464=1126.981,260.706,-71.176,-178.405,10.027,149.563
C02465=1126.977,260.955,-71.204,-178.402,10.029,149.563
C02466=1126.972,261.203,-71.234,-178.398,10.033,149.563
C02467=1126.968,261.451,-71.263,-178.395,10.035,149.562
C02468=1126.964,261.699,-71.291,-178.391,10.039,149.562
C02469=1126.960,261.948,-71.320,-178.388,10.042,149.562
C02470=1126.956,262.196,-71.350,-178.384,10.045,149.562
C02471=1126.951,262.445,-71.379,-178.381,10.048,149.562
C02472=1126.947,262.692,-71.407,-178.377,10.051,149.562
C02473=1126.943,262.940,-71.437,-178.373,10.054,149.561
C02474=1126.938,263.189,-71.465,-178.370,10.057,149.561
C02475=1126.934,263.437,-71.495,-178.366,10.060,149.561
C02476=1126.930,263.686,-71.524,-178.362,10.063,149.561
C02477=1126.925,263.934,-71.553,-178.359,10.067,149.561
C02478=1126.921,264.182,-71.582,-178.355,10.070,149.560
C02479=1126.916,264.430,-71.612,-178.351,10.073,149.560
C02480=1126.913,264.678,-71.640,-178.349,10.075,149.560
C02481=1126.909,264.927,-71.670,-178.346,10.078,149.560
C02482=1126.904,265.176,-71.699,-178.343,10.080,149.560
C02483=1126.900,265.424,-71.728,-178.341,10.082,149.560
C02484=1126.895,265.671,-71.757,-178.338,10.085,149.560
C02485=1126.891,265.920,-71.787,-178.336,10.087,149.559
C02486=1126.887,266.168,-71.816,-178.333,10.090,149.559
C02487=1126.883,266.381,-71.841,-178.331,10.091,149.559
C02488=1126.880,266.595,-71.866,-178.329,10.093,149.559
C02489=1126.876,266.808,-71.892,-178.327,10.096,149.559
C02490=1126.872,267.022,-71.917,-178.324,10.098,149.559
C02491=1126.868,267.236,-71.942,-178.322,10.100,149.559
C02492=1126.865,267.449,-71.967,-178.320,10.102,149.559
C02493=1126.862,267.664,-71.993,-178.317,10.104,149.559
C02494=1126.858,267.877,-72.018,-178.316,10.106,149.559
C02495=1126.854,268.125,-72.047,-178.313,10.109,149.559
C02496=1126.849,268.373,-72.076,-178.310,10.111,149.559
C02497=1126.845,268.621,-72.106,-178.307,10.114,149.558
C02498=1126.841,268.869,-72.135,-178.305,10.116,149.558
C02499=1126.837,269.118,-72.165,-178.302,10.118,149.558
C02500=1126.832,269.366,-72.194,-178.299,10.121,149.558
C02501=1126.828,269.614,-72.224,-178.296,10.124,149.558
C02502=1126.823,269.863,-72.254,-178.294,10.126,149.558
C02503=1126.819,270.110,-72.284,-178.291,10.129,149.558
C02504=1126.815,270.359,-72.313,-178.288,10.131,149.558
C02505=1126.811,270.607,-72.343,-178.285,10.134,149.558
C02506=1126.807,270.855,-72.372,-178.283,10.136,149.557
C02507=1126.803,271.103,-72.402,-178.280,10.139,149.557
C02508=1126.799,271.352,-72.431,-178.277,10.142,149.557
C02509=1126.794,271.600,-72.460,-178.274,10.144,149.557
C02510=1126.790,271.848,-72.490,-178.271,10.147,149.557
C02511=1126.786,272.096,-72.520,-178.268,10.150,149.557
C02512=1126.781,272.344,-72.550,-178.266,10.152,149.557
C02513=1126.777,272.593,-72.580,-178.263,10.155,149.557
C02514=1126.773,272.841,-72.609,-178.260,10.157,149.556
C02515=1126.769,273.089,-72.638,-178.257,10.160,149.556
C02516=1126.765,273.337,-72.669,-178.254,10.163,149.556
C02517=1126.761,273.585,-72.698,-178.251,10.165,149.556
C02518=1126.756,273.834,-72.728,-178.248,10.168,149.556
C02519=1126.752,274.081,-72.758,-178.245,10.171,149.556
C02520=1126.748,274.330,-72.788,-178.241,10.173,149.556
C02521=1126.744,274.578,-72.817,-178.239,10.176,149.556
C02522=1126.739,274.826,-72.847,-178.236,10.179,149.555
C02523=1126.735,275.074,-72.877,-178.233,10.181,149.555
C02524=1126.731,275.322,-72.907,-178.230,10.184,149.555
C02525=1126.727,275.571,-72.937,-178.226,10.187,149.555
C02526=1126.723,275.819,-72.967,-178.223,10.189,149.555
C02527=1126.718,276.068,-72.997,-178.220,10.193,149.555
C02528=1126.714,276.315,-73.027,-178.217,10.195,149.554
C02529=1126.710,276.564,-73.057,-178.214,10.198,149.554
C02530=1126.706,276.811,-73.087,-178.211,10.201,149.554
C02531=1126.701,277.060,-73.117,-178.207,10.203,149.554
C02532=1126.698,277.307,-73.147,-178.204,10.206,149.554
C02533=1126.693,277.556,-73.177,-178.200,10.209,149.554
C02534=1126.689,277.804,-73.208,-178.197,10.212,149.554
C02535=1126.685,278.053,-73.237,-178.195,10.215,149.553
C02536=1126.681,278.301,-73.268,-178.191,10.217,149.553
C02537=1126.676,278.549,-73.297,-178.188,10.220,149.553
C02538=1126.672,278.796,-73.327,-178.184,10.223,149.553
C02539=1126.668,279.045,-73.357,-178.181,10.226,149.553
C02540=1126.664,279.293,-73.388,-178.178,10.228,149.552
C02541=1126.660,279.541,-73.418,-178.174,10.231,149.552
C02542=1126.655,279.790,-73.448,-178.171,10.234,149.552
C02543=1126.652,280.002,-73.474,-178.168,10.237,149.552
C02544=1126.648,280.216,-73.500,-178.165,10.239,149.552
C02545=1126.645,280.430,-73.527,-178.162,10.241,149.552
C02546=1126.641,280.643,-73.553,-178.159,10.244,149.551
C02547=1126.637,280.856,-73.578,-178.156,10.247,149.551
C02548=1126.634,281.069,-73.604,-178.153,10.248,149.551
C02549=1126.630,281.284,-73.630,-178.151,10.251,149.551
C02550=1126.627,281.497,-73.656,-178.147,10.253,149.550
C02551=1126.622,281.744,-73.687,-178.144,10.256,149.550
C02552=1126.619,281.993,-73.718,-178.141,10.259,149.550
C02553=1126.614,282.241,-73.748,-178.138,10.261,149.550
C02554=1126.610,282.489,-73.778,-178.135,10.264,149.550
C02555=1126.605,282.737,-73.809,-178.132,10.266,149.550
C02556=1126.601,282.985,-73.839,-178.129,10.268,149.550
C02557=1126.598,283.233,-73.870,-178.126,10.271,149.549
C02558=1126.593,283.481,-73.901,-178.123,10.274,149.549
C02559=1126.589,283.730,-73.930,-178.120,10.276,149.549
C02560=1126.585,283.978,-73.961,-178.117,10.279,149.549
C02561=1126.581,284.226,-73.991,-178.114,10.282,149.549
C02562=1126.576,284.474,-74.022,-178.111,10.284,149.548
C02563=1126.572,284.722,-74.053,-178.108,10.287,149.548
C02564=1126.568,284.970,-74.083,-178.104,10.289,149.548
C02565=1126.564,285.218,-74.114,-178.102,10.291,149.548
C02566=1126.560,285.466,-74.144,-178.099,10.294,149.548
C02567=1126.556,285.714,-74.176,-178.096,10.296,149.548
C02568=1126.551,285.962,-74.206,-178.093,10.299,149.547
C02569=1126.547,286.210,-74.236,-178.089,10.302,149.547
C02570=1126.543,286.458,-74.267,-178.086,10.304,149.547
C02571=1126.539,286.707,-74.298,-178.083,10.307,149.547
C02572=1126.535,286.954,-74.329,-178.080,10.310,149.547
C02573=1126.530,287.202,-74.359,-178.077,10.312,149.546
C02574=1126.526,287.451,-74.390,-178.074,10.315,149.546
C02575=1126.522,287.699,-74.421,-178.071,10.316,149.546
C02576=1126.518,287.947,-74.452,-178.068,10.319,149.546
C02577=1126.514,288.195,-74.482,-178.065,10.322,149.546
C02578=1126.509,288.443,-74.513,-178.062,10.324,149.546
C02579=1126.506,288.691,-74.544,-178.059,10.327,149.545
C02580=1126.502,288.939,-74.575,-178.056,10.329,149.545
C02581=1126.497,289.187,-74.606,-178.053,10.332,149.545
C02582=1126.493,289.435,-74.637,-178.049,10.335,149.545
C02583=1126.488,289.683,-74.668,-178.046,10.337,149.545
C02584=1126.485,289.932,-74.698,-178.043,10.340,149.544
C02585=1126.481,290.179,-74.730,-178.040,10.343,149.544
C02586=1126.476,290.427,-74.761,-178.038,10.344,149.544
C02587=1126.472,290.676,-74.792,-178.035,10.347,149.544
C02588=1126.468,290.924,-74.823,-178.032,10.350,149.544
C02589=1126.465,291.171,-74.854,-178.028,10.352,149.544
C02590=1126.460,291.419,-74.885,-178.025,10.355,149.544
C02591=1126.456,291.668,-74.916,-178.022,10.357,149.543
C02592=1126.452,291.915,-74.947,-178.019,10.360,149.543
C02593=1126.448,292.164,-74.978,-178.016,10.363,149.543
C02594=1126.443,292.412,-75.009,-178.013,10.365,149.543
C02595=1126.439,292.659,-75.040,-178.009,10.368,149.543
C02596=1126.435,292.908,-75.071,-178.007,10.371,149.542
C02597=1126.431,293.156,-75.102,-178.004,10.372,149.542
C02598=1126.427,293.404,-75.134,-178.001,10.375,149.542
C02599=1126.423,293.617,-75.160,-177.998,10.378,149.542
C02600=1126.420,293.831,-75.187,-177.995,10.379,149.542
C02601=1126.416,294.043,-75.214,-177.993,10.381,149.542
C02602=1126.413,294.257,-75.241,-177.990,10.384,149.541
C02603=1126.409,294.470,-75.268,-177.988,10.386,149.541
C02604=1126.406,294.683,-75.295,-177.984,10.389,149.541
C02605=1126.402,294.897,-75.322,-177.982,10.390,149.541
C02606=1126.398,295.110,-75.349,-177.980,10.392,149.541
C02607=1126.394,295.358,-75.380,-177.976,10.395,149.541
C02608=1126.390,295.606,-75.411,-177.974,10.398,149.541
C02609=1126.386,295.854,-75.443,-177.970,10.400,149.540
C02610=1126.381,296.102,-75.474,-177.967,10.403,149.540
C02611=1126.378,296.350,-75.506,-177.964,10.405,149.540
C02612=1126.373,296.597,-75.537,-177.961,10.408,149.540
C02613=1126.369,296.846,-75.568,-177.958,10.410,149.540
C02614=1126.365,297.093,-75.600,-177.955,10.413,149.539
C02615=1126.361,297.342,-75.631,-177.952,10.415,149.539
C02616=1126.357,297.590,-75.663,-177.949,10.418,149.539
C02617=1126.353,297.837,-75.694,-177.946,10.420,149.539
C02618=1126.349,298.086,-75.725,-177.943,10.423,149.539
C02619=1126.345,298.333,-75.757,-177.939,10.425,149.538
C02620=1126.341,298.581,-75.789,-177.937,10.428,149.538
C02621=1126.336,298.829,-75.819,-177.933,10.430,149.538
C02622=1126.333,299.077,-75.851,-177.930,10.433,149.538
C02623=1126.328,299.326,-75.884,-177.927,10.436,149.538
C02624=1126.324,299.573,-75.915,-177.924,10.438,149.538
C02625=1126.320,299.822,-75.946,-177.921,10.441,149.537
C02626=1126.316,300.069,-75.978,-177.918,10.444,149.537
C02627=1126.312,300.317,-76.010,-177.914,10.446,149.537
C02628=1126.308,300.565,-76.041,-177.912,10.448,149.537
C02629=1126.304,300.813,-76.073,-177.909,10.450,149.537
C02630=1126.299,301.062,-76.105,-177.906,10.453,149.537
C02631=1126.296,301.310,-76.136,-177.902,10.456,149.536
C02632=1126.291,301.557,-76.168,-177.900,10.458,149.536
C02633=1126.288,301.805,-76.200,-177.896,10.461,149.536
C02634=1126.283,302.053,-76.232,-177.893,10.464,149.536
C02635=1126.279,302.301,-76.264,-177.890,10.466,149.536
C02636=1126.275,302.549,-76.296,-177.887,10.469,149.536
C02637=1126.271,302.797,-76.327,-177.884,10.471,149.535
C02638=1126.266,303.044,-76.360,-177.880,10.474,149.535
C02639=1126.263,303.292,-76.391,-177.877,10.476,149.535
C02640=1126.259,303.540,-76.423,-177.875,10.478,149.535
C02641=1126.255,303.788,-76.455,-177.872,10.481,149.535
C02642=1126.250,304.036,-76.487,-177.868,10.483,149.534
C02643=1126.246,304.284,-76.519,-177.866,10.486,149.534
C02644=1126.242,304.532,-76.550,-177.862,10.489,149.534
C02645=1126.238,304.780,-76.583,-177.859,10.491,149.534
C02646=1126.234,305.028,-76.615,-177.856,10.494,149.534
C02647=1126.230,305.276,-76.647,-177.853,10.497,149.534
C02648=1126.225,305.524,-76.679,-177.850,10.499,149.533
C02649=1126.222,305.772,-76.710,-177.847,10.502,149.533
C02650=1126.217,306.020,-76.743,-177.843,10.504,149.533
C02651=1126.213,306.267,-76.774,-177.840,10.507,149.533
C02652=1126.209,306.515,-76.806,-177.837,10.509,149.533
C02653=1126.205,306.763,-76.839,-177.834,10.512,149.532
C02654=1126.201,307.011,-76.871,-177.832,10.514,149.532
C02655=1126.198,307.224,-76.898,-177.828,10.516,149.532
C02656=1126.194,307.437,-76.927,-177.826,10.518,149.532
C02657=1126.191,307.650,-76.954,-177.823,10.521,149.532
C02658=1126.188,307.864,-76.982,-177.820,10.523,149.531
C02659=1126.183,308.076,-77.010,-177.818,10.525,149.531
C02660=1126.180,308.289,-77.037,-177.815,10.527,149.531
C02661=1126.176,308.503,-77.065,-177.812,10.529,149.531
C02662=1126.173,308.716,-77.093,-177.810,10.531,149.531
C02663=1126.169,308.964,-77.124,-177.807,10.534,149.531
C02664=1126.164,309.212,-77.157,-177.804,10.536,149.531
C02665=1126.161,309.460,-77.189,-177.800,10.539,149.530
C02666=1126.156,309.708,-77.222,-177.798,10.541,149.530
C02667=1126.153,309.956,-77.254,-177.794,10.544,149.530
C02668=1126.149,310.203,-77.287,-177.791,10.547,149.530
C02669=1126.144,310.451,-77.318,-177.788,10.549,149.530
C02670=1126.140,310.699,-77.351,-177.785,10.552,149.530
C02671=1126.136,310.947,-77.383,-177.782,10.554,149.529
C02672=1126.132,311.195,-77.416,-177.778,10.557,149.529
C02673=1126.128,311.443,-77.449,-177.775,10.560,149.529
C02674=1126.124,311.691,-77.481,-177.772,10.562,149.529
C02675=1126.120,311.939,-77.513,-177.769,10.565,149.529
C02676=1126.116,312.186,-77.545,-177.766,10.566,149.528
C02677=1126.111,312.434,-77.578,-177.763,10.569,149.528
C02678=1126.108,312.681,-77.610,-177.760,10.572,149.528
C02679=1126.103,312.930,-77.643,-177.757,10.574,149.528
C02680=1126.099,313.178,-77.676,-177.754,10.577,149.528
C02681=1126.096,313.426,-77.708,-177.751,10.579,149.527
C02682=1126.091,313.673,-77.741,-177.747,10.582,149.527
C02683=1126.087,313.921,-77.774,-177.744,10.584,149.527
C02684=1126.084,314.169,-77.806,-177.741,10.587,149.527
C02685=1126.080,314.417,-77.839,-177.738,10.590,149.527
C02686=1126.075,314.665,-77.872,-177.735,10.592,149.527
C02687=1126.072,314.913,-77.904,-177.731,10.595,149.526
C02688=1126.068,315.160,-77.937,-177.729,10.597,149.526
C02689=1126.063,315.409,-77.970,-177.725,10.600,149.526
C02690=1126.059,315.655,-78.002,-177.722,10.603,149.526
C02691=1126.055,315.903,-78.035,-177.720,10.604,149.526
C02692=1126.051,316.151,-78.068,-177.716,10.607,149.525
C02693=1126.047,316.399,-78.100,-177.713,10.609,149.525
C02694=1126.043,316.647,-78.133,-177.710,10.612,149.525
C02695=1126.039,316.894,-78.166,-177.707,10.615,149.525
C02696=1126.034,317.143,-78.199,-177.704,10.617,149.525
C02697=1126.031,317.390,-78.231,-177.700,10.619,149.524
C02698=1126.027,317.638,-78.265,-177.697,10.622,149.524
C02699=1126.023,317.886,-78.298,-177.694,10.625,149.524
C02700=1126.018,318.134,-78.330,-177.691,10.627,149.524
C02701=1126.015,318.381,-78.363,-177.688,10.630,149.524
C02702=1126.011,318.630,-78.396,-177.685,10.632,149.524
C02703=1126.007,318.878,-78.429,-177.682,10.635,149.523
C02704=1126.003,319.125,-78.463,-177.678,10.638,149.523
C02705=1125.999,319.373,-78.496,-177.675,10.640,149.523
C02706=1125.995,319.621,-78.529,-177.672,10.643,149.523
C02707=1125.991,319.868,-78.561,-177.669,10.644,149.523
C02708=1125.987,320.116,-78.594,-177.666,10.647,149.522
C02709=1125.983,320.364,-78.627,-177.663,10.650,149.522
C02710=1125.979,320.612,-78.660,-177.660,10.652,149.522
C02711=1125.975,320.825,-78.689,-177.657,10.655,149.522
C02712=1125.972,321.037,-78.717,-177.654,10.657,149.522
C02713=1125.969,321.251,-78.746,-177.652,10.659,149.522
C02714=1125.965,321.464,-78.774,-177.649,10.661,149.521
C02715=1125.961,321.677,-78.803,-177.646,10.663,149.521
C02716=1125.958,321.890,-78.831,-177.643,10.666,149.521
C02717=1125.955,322.103,-78.860,-177.641,10.667,149.521
C02718=1125.951,322.316,-78.889,-177.638,10.669,149.521
C02719=1125.947,322.563,-78.922,-177.635,10.672,149.521
C02720=1125.943,322.811,-78.955,-177.632,10.674,149.520
C02721=1125.939,323.059,-78.988,-177.629,10.677,149.520
C02722=1125.935,323.307,-79.021,-177.625,10.680,149.520
C02723=1125.931,323.554,-79.054,-177.622,10.682,149.520
C02724=1125.928,323.802,-79.087,-177.619,10.685,149.520
C02725=1125.924,324.049,-79.121,-177.616,10.687,149.519
C02726=1125.919,324.298,-79.155,-177.613,10.690,149.519
C02727=1125.915,324.545,-79.188,-177.610,10.692,149.519
C02728=1125.911,324.793,-79.221,-177.606,10.695,149.519
C02729=1125.907,325.041,-79.254,-177.603,10.697,149.519
C02730=1125.903,325.288,-79.288,-177.600,10.700,149.519
C02731=1125.899,325.536,-79.322,-177.597,10.703,149.518
C02732=1125.895,325.784,-79.355,-177.593,10.705,149.518
C02733=1125.891,326.032,-79.388,-177.591,10.707,149.518
C02734=1125.887,326.279,-79.422,-177.588,10.709,149.518
C02735=1125.883,326.527,-79.455,-177.584,10.712,149.518
C02736=1125.880,326.775,-79.489,-177.582,10.715,149.517
C02737=1125.876,327.022,-79.523,-177.578,10.717,149.517
C02738=1125.872,327.270,-79.556,-177.575,10.720,149.517
C02739=1125.867,327.518,-79.589,-177.572,10.722,149.517
C02740=1125.863,327.765,-79.623,-177.569,10.725,149.517
C02741=1125.859,328.013,-79.657,-177.565,10.727,149.516
C02742=1125.855,328.261,-79.690,-177.562,10.730,149.516
C02743=1125.851,328.508,-79.724,-177.559,10.732,149.516
C02744=1125.847,328.756,-79.757,-177.556,10.735,149.516
C02745=1125.844,329.004,-79.791,-177.552,10.737,149.516
C02746=1125.839,329.252,-79.825,-177.550,10.740,149.516
C02747=1125.835,329.499,-79.859,-177.546,10.743,149.515
C02748=1125.831,329.747,-79.892,-177.543,10.745,149.515
C02749=1125.828,329.994,-79.926,-177.540,10.747,149.515
C02750=1125.824,330.242,-79.959,-177.537,10.750,149.515
C02751=1125.819,330.490,-79.994,-177.534,10.752,149.514
C02752=1125.816,330.738,-80.027,-177.531,10.754,149.514
C02753=1125.812,330.985,-80.061,-177.528,10.757,149.514
C02754=1125.808,331.233,-80.094,-177.524,10.760,149.514
C02755=1125.803,331.480,-80.129,-177.521,10.762,149.514
C02756=1125.800,331.729,-80.162,-177.518,10.764,149.513
C02757=1125.796,331.976,-80.196,-177.515,10.767,149.513
C02758=1125.791,332.223,-80.231,-177.512,10.770,149.513
C02759=1125.788,332.472,-80.264,-177.508,10.772,149.513
C02760=1125.784,332.719,-80.298,-177.505,10.775,149.513
C02761=1125.779,332.966,-80.333,-177.502,10.777,149.513
C02762=1125.776,333.215,-80.366,-177.499,10.780,149.512
C02763=1125.772,333.462,-80.400,-177.495,10.782,149.512
C02764=1125.767,333.709,-80.434,-177.492,10.785,149.512
C02765=1125.764,333.958,-80.468,-177.489,10.788,149.512
C02766=1125.760,334.205,-80.502,-177.486,10.790,149.512
C02767=1125.756,334.418,-80.531,-177.483,10.792,149.512
C02768=1125.754,334.631,-80.561,-177.481,10.794,149.511
C02769=1125.750,334.844,-80.590,-177.478,10.796,149.511
C02770=1125.746,335.056,-80.620,-177.475,10.798,149.511
C02771=1125.743,335.269,-80.649,-177.472,10.801,149.511
C02772=1125.739,335.482,-80.678,-177.470,10.803,149.511
C02773=1125.736,335.694,-80.707,-177.467,10.804,149.510
C02774=1125.733,335.908,-80.736,-177.464,10.807,149.510
C02775=1125.729,336.155,-80.771,-177.461,10.809,149.510
C02776=1125.725,336.403,-80.805,-177.457,10.812,149.510
C02777=1125.721,336.650,-80.840,-177.454,10.815,149.510
C02778=1125.717,336.897,-80.873,-177.451,10.817,149.509
C02779=1125.713,337.145,-80.908,-177.448,10.820,149.509
C02780=1125.709,337.393,-80.941,-177.445,10.821,149.509
C02781=1125.705,337.641,-80.976,-177.442,10.824,149.509
C02782=1125.701,337.888,-81.010,-177.439,10.827,149.509
C02783=1125.697,338.137,-81.045,-177.436,10.829,149.508
C02784=1125.693,338.384,-81.079,-177.432,10.831,149.508
C02785=1125.689,338.631,-81.113,-177.429,10.834,149.508
C02786=1125.685,338.879,-81.148,-177.426,10.837,149.508
C02787=1125.681,339.126,-81.182,-177.423,10.839,149.508
C02788=1125.678,339.374,-81.216,-177.419,10.842,149.507
C02789=1125.673,339.622,-81.251,-177.416,10.844,149.507
C02790=1125.670,339.869,-81.285,-177.413,10.846,149.507
C02791=1125.666,340.116,-81.320,-177.410,10.849,149.507
C02792=1125.662,340.364,-81.355,-177.406,10.852,149.507
C02793=1125.658,340.611,-81.389,-177.403,10.854,149.506
C02794=1125.654,340.859,-81.424,-177.400,10.857,149.506
C02795=1125.649,341.107,-81.458,-177.397,10.859,149.506
C02796=1125.646,341.355,-81.492,-177.394,10.862,149.506
C02797=1125.641,341.602,-81.527,-177.390,10.864,149.506
C02798=1125.639,341.849,-81.562,-177.387,10.867,149.505
C02799=1125.634,342.097,-81.596,-177.384,10.868,149.505
C02800=1125.630,342.345,-81.631,-177.381,10.871,149.505
C02801=1125.625,342.592,-81.666,-177.378,10.874,149.505
C02802=1125.622,342.840,-81.700,-177.375,10.876,149.505
C02803=1125.618,343.087,-81.735,-177.371,10.879,149.504
C02804=1125.614,343.335,-81.770,-177.368,10.881,149.504
C02805=1125.611,343.583,-81.804,-177.365,10.884,149.504
C02806=1125.606,343.830,-81.839,-177.361,10.886,149.504
C02807=1125.603,344.078,-81.874,-177.359,10.889,149.504
C02808=1125.598,344.325,-81.909,-177.355,10.891,149.504
C02809=1125.595,344.573,-81.943,-177.352,10.894,149.503
C02810=1125.590,344.820,-81.978,-177.349,10.896,149.503
C02811=1125.586,345.068,-82.013,-177.345,10.899,149.503
C02812=1125.583,345.315,-82.048,-177.342,10.901,149.503
C02813=1125.579,345.563,-82.082,-177.339,10.904,149.503
C02814=1125.575,345.811,-82.117,-177.336,10.906,149.502
C02815=1125.571,346.057,-82.152,-177.332,10.909,149.502
C02816=1125.567,346.306,-82.187,-177.329,10.911,149.502
C02817=1125.563,346.553,-82.223,-177.326,10.914,149.502
C02818=1125.559,346.800,-82.256,-177.323,10.916,149.501
C02819=1125.556,347.048,-82.292,-177.320,10.918,149.501
C02820=1125.552,347.296,-82.327,-177.317,10.921,149.501
C02821=1125.547,347.543,-82.362,-177.314,10.923,149.501
C02822=1125.543,347.791,-82.397,-177.310,10.926,149.501
C02823=1125.540,348.003,-82.426,-177.307,10.928,149.500
C02824=1125.537,348.216,-82.457,-177.305,10.930,149.500
C02825=1125.534,348.428,-82.487,-177.301,10.932,149.500
C02826=1125.530,348.642,-82.517,-177.299,10.934,149.500
C02827=1125.527,348.854,-82.547,-177.296,10.936,149.500
C02828=1125.523,349.066,-82.578,-177.293,10.939,149.500
C02829=1125.520,349.279,-82.608,-177.291,10.941,149.499
C02830=1125.517,349.492,-82.638,-177.287,10.943,149.499
C02831=1125.513,349.740,-82.673,-177.284,10.946,149.499
C02832=1125.509,349.987,-82.708,-177.281,10.948,149.499
C02833=1125.505,350.234,-82.743,-177.277,10.951,149.498
C02834=1125.501,350.482,-82.778,-177.273,10.953,149.498
C02835=1125.497,350.730,-82.814,-177.270,10.956,149.498
C02836=1125.494,350.977,-82.849,-177.267,10.958,149.498
C02837=1125.489,351.224,-82.885,-177.263,10.962,149.498
C02838=1125.485,351.472,-82.919,-177.259,10.964,149.497
C02839=1125.482,351.719,-82.955,-177.256,10.966,149.497
C02840=1125.478,351.967,-82.990,-177.252,10.969,149.497
C02841=1125.474,352.214,-83.026,-177.248,10.972,149.496
C02842=1125.470,352.461,-83.061,-177.245,10.974,149.496
C02843=1125.466,352.709,-83.096,-177.241,10.976,149.496
C02844=1125.463,352.957,-83.132,-177.237,10.980,149.496
C02845=1125.458,353.204,-83.167,-177.234,10.982,149.495
C02846=1125.455,353.451,-83.202,-177.231,10.985,149.495
C02847=1125.451,353.699,-83.238,-177.228,10.987,149.495
C02848=1125.447,353.946,-83.273,-177.224,10.989,149.495
C02849=1125.444,354.194,-83.309,-177.220,10.992,149.494
C02850=1125.439,354.440,-83.344,-177.217,10.995,149.494
C02851=1125.436,354.688,-83.380,-177.213,10.997,149.494
C02852=1125.431,354.936,-83.416,-177.210,10.999,149.494
C02853=1125.428,355.183,-83.451,-177.206,11.002,149.493
C02854=1125.424,355.431,-83.487,-177.203,11.004,149.493
C02855=1125.420,355.678,-83.522,-177.199,11.008,149.493
C02856=1125.417,355.926,-83.558,-177.195,11.010,149.492
C02857=1125.412,356.173,-83.593,-177.192,11.012,149.492
C02858=1125.409,356.420,-83.629,-177.189,11.015,149.492
C02859=1125.404,356.668,-83.665,-177.185,11.017,149.492
C02860=1125.401,356.915,-83.700,-177.182,11.019,149.491
C02861=1125.397,357.163,-83.736,-177.178,11.022,149.491
C02862=1125.393,357.410,-83.772,-177.175,11.024,149.491
C02863=1125.390,357.658,-83.807,-177.171,11.027,149.491
C02864=1125.386,357.905,-83.844,-177.167,11.030,149.490
C02865=1125.381,358.152,-83.879,-177.164,11.032,149.490
C02866=1125.378,358.399,-83.915,-177.161,11.035,149.490
C02867=1125.374,358.647,-83.950,-177.157,11.037,149.490
C02868=1125.370,358.895,-83.986,-177.154,11.039,149.489
C02869=1125.366,359.142,-84.023,-177.150,11.042,149.489
C02870=1125.363,359.389,-84.058,-177.147,11.044,149.489
C02871=1125.359,359.637,-84.094,-177.144,11.047,149.489
C02872=1125.355,359.884,-84.130,-177.140,11.049,149.488
C02873=1125.351,360.131,-84.166,-177.137,11.051,149.488
C02874=1125.348,360.379,-84.202,-177.134,11.054,149.488
C02875=1125.343,360.627,-84.238,-177.130,11.056,149.488
C02876=1125.340,360.873,-84.274,-177.127,11.058,149.487
C02877=1125.336,361.121,-84.310,-177.123,11.061,149.487
C02878=1125.332,361.369,-84.346,-177.120,11.063,149.487
C02879=1125.329,361.581,-84.377,-177.117,11.066,149.487
C02880=1125.326,361.793,-84.407,-177.114,11.067,149.486
C02881=1125.323,362.006,-84.439,-177.111,11.069,149.486
C02882=1125.320,362.218,-84.470,-177.108,11.071,149.486
C02883=1125.316,362.430,-84.501,-177.106,11.074,149.486
C02884=1125.313,362.644,-84.531,-177.102,11.076,149.486
C02885=1125.310,362.856,-84.563,-177.100,11.078,149.485
C02886=1125.306,363.068,-84.594,-177.097,11.079,149.485
C02887=1125.302,363.315,-84.630,-177.094,11.082,149.485
C02888=1125.298,363.563,-84.666,-177.090,11.084,149.484
C02889=1125.295,363.810,-84.702,-177.087,11.086,149.484
C02890=1125.290,364.058,-84.738,-177.083,11.089,149.484
C02891=1125.287,364.304,-84.775,-177.080,11.091,149.484
C02892=1125.283,364.553,-84.811,-177.077,11.094,149.484
C02893=1125.280,364.800,-84.847,-177.073,11.096,149.483
C02894=1125.276,365.048,-84.884,-177.070,11.098,149.483
C02895=1125.272,365.295,-84.920,-177.066,11.101,149.483
C02896=1125.268,365.542,-84.957,-177.063,11.103,149.483
C02897=1125.264,365.789,-84.992,-177.060,11.106,149.482
C02898=1125.260,366.036,-85.029,-177.057,11.108,149.482
C02899=1125.257,366.283,-85.065,-177.054,11.110,149.482
C02900=1125.253,366.531,-85.101,-177.051,11.113,149.482
C02901=1125.249,366.778,-85.138,-177.047,11.115,149.481
C02902=1125.245,367.025,-85.175,-177.044,11.117,149.481
C02903=1125.241,367.273,-85.211,-177.040,11.120,149.481
C02904=1125.237,367.520,-85.247,-177.037,11.122,149.481
C02905=1125.234,367.768,-85.284,-177.034,11.125,149.480
C02906=1125.231,368.015,-85.321,-177.030,11.127,149.480
C02907=1125.226,368.262,-85.357,-177.028,11.129,149.480
C02908=1125.222,368.510,-85.394,-177.024,11.131,149.480
C02909=1125.219,368.757,-85.430,-177.021,11.134,149.480
C02910=1125.215,369.004,-85.467,-177.018,11.136,149.479
C02911=1125.211,369.251,-85.503,-177.015,11.139,149.479
C02912=1125.208,369.499,-85.540,-177.011,11.141,149.479
C02913=1125.203,369.746,-85.576,-177.009,11.143,149.479
C02914=1125.200,369.993,-85.613,-177.005,11.145,149.478
C02915=1125.196,370.240,-85.649,-177.002,11.148,149.478
C02916=1125.192,370.488,-85.686,-176.999,11.150,149.478
C02917=1125.188,370.734,-85.722,-176.995,11.153,149.478
C02918=1125.185,370.982,-85.760,-176.993,11.154,149.478
C02919=1125.181,371.230,-85.797,-176.989,11.157,149.477
C02920=1125.177,371.476,-85.833,-176.986,11.159,149.477
C02921=1125.173,371.724,-85.870,-176.983,11.162,149.477
C02922=1125.169,371.971,-85.907,-176.979,11.164,149.477
C02923=1125.166,372.219,-85.944,-176.977,11.166,149.477
C02924=1125.162,372.466,-85.980,-176.974,11.169,149.476
C02925=1125.158,372.713,-86.017,-176.970,11.171,149.476
C02926=1125.154,372.960,-86.054,-176.967,11.173,149.476
C02927=1125.150,373.207,-86.091,-176.964,11.176,149.476
C02928=1125.147,373.455,-86.127,-176.961,11.178,149.476
C02929=1125.143,373.702,-86.164,-176.958,11.180,149.475
C02930=1125.139,373.949,-86.201,-176.955,11.183,149.475
C02931=1125.135,374.196,-86.238,-176.951,11.185,149.475
C02932=1125.132,374.444,-86.276,-176.949,11.187,149.475
C02933=1125.129,374.690,-86.312,-176.945,11.190,149.475
C02934=1125.124,374.938,-86.349,-176.943,11.192,149.475
C02935=1125.121,375.151,-86.381,-176.940,11.194,149.474
C02936=1125.118,375.363,-86.413,-176.938,11.196,149.474
C02937=1125.115,375.575,-86.444,-176.934,11.199,149.474
C02938=1125.111,375.788,-86.477,-176.932,11.201,149.474
C02939=1125.108,376.000,-86.508,-176.929,11.202,149.474
C02940=1125.106,376.212,-86.540,-176.927,11.204,149.474
C02941=1125.101,376.425,-86.571,-176.924,11.206,149.473
C02942=1125.099,376.637,-86.603,-176.922,11.209,149.473
C02943=1125.095,376.884,-86.641,-176.919,11.211,149.473
C02944=1125.091,377.131,-86.678,-176.916,11.213,149.473
C02945=1125.087,377.378,-86.715,-176.913,11.216,149.473
C02946=1125.084,377.626,-86.752,-176.910,11.218,149.473
C02947=1125.080,377.873,-86.790,-176.907,11.220,149.473
C02948=1125.076,378.120,-86.827,-176.904,11.223,149.473
C02949=1125.072,378.367,-86.864,-176.901,11.225,149.472
C02950=1125.068,378.614,-86.901,-176.898,11.227,149.472
C02951=1125.064,378.862,-86.938,-176.895,11.230,149.472
C02952=1125.061,379.109,-86.976,-176.892,11.233,149.472
C02953=1125.058,379.356,-87.013,-176.889,11.234,149.472
C02954=1125.054,379.603,-87.049,-176.887,11.237,149.472
C02955=1125.051,379.850,-87.087,-176.883,11.240,149.472
C02956=1125.046,380.097,-87.124,-176.880,11.242,149.472
C02957=1125.043,380.344,-87.162,-176.878,11.244,149.471
C02958=1125.039,380.592,-87.199,-176.875,11.247,149.471
C02959=1125.034,380.839,-87.236,-176.871,11.249,149.471
C02960=1125.031,381.086,-87.274,-176.869,11.251,149.471
C02961=1125.027,381.334,-87.311,-176.866,11.254,149.471
C02962=1125.023,381.580,-87.349,-176.863,11.257,149.471
C02963=1125.020,381.828,-87.387,-176.861,11.259,149.471
C02964=1125.016,382.075,-87.424,-176.857,11.261,149.471
C02965=1125.013,382.322,-87.462,-176.855,11.264,149.471
C02966=1125.009,382.569,-87.498,-176.852,11.266,149.471
C02967=1125.005,382.816,-87.536,-176.849,11.269,149.471
C02968=1125.001,383.064,-87.573,-176.846,11.271,149.470
C02969=1124.998,383.310,-87.611,-176.843,11.274,149.470
C02970=1124.994,383.558,-87.649,-176.841,11.276,149.470
C02971=1124.990,383.805,-87.686,-176.840,11.278,149.470
C02972=1124.987,384.052,-87.724,-176.838,11.280,149.470
C02973=1124.983,384.299,-87.762,-176.836,11.281,149.470
C02974=1124.979,384.546,-87.799,-176.834,11.284,149.471
C02975=1124.975,384.793,-87.836,-176.833,11.285,149.471
C02976=1124.972,385.040,-87.874,-176.831,11.288,149.471
C02977=1124.968,385.288,-87.911,-176.829,11.290,149.471
C02978=1124.964,385.534,-87.949,-176.828,11.291,149.471
C02979=1124.961,385.782,-87.987,-176.826,11.294,149.471
C02980=1124.957,386.029,-88.025,-176.824,11.295,149.471
C02981=1124.953,386.276,-88.062,-176.823,11.298,149.471
C02982=1124.949,386.523,-88.100,-176.821,11.300,149.471
C02983=1124.946,386.770,-88.138,-176.820,11.302,149.472
C02984=1124.942,387.017,-88.175,-176.818,11.304,149.472
C02985=1124.939,387.265,-88.213,-176.816,11.307,149.472
C02986=1124.934,387.512,-88.251,-176.815,11.308,149.472
C02987=1124.931,387.759,-88.289,-176.813,11.311,149.472
C02988=1124.927,388.005,-88.326,-176.812,11.313,149.472
C02989=1124.924,388.253,-88.363,-176.810,11.315,149.472
C02990=1124.920,388.500,-88.401,-176.809,11.318,149.473
C02991=1124.917,388.712,-88.434,-176.808,11.319,149.473
C02992=1124.913,388.925,-88.466,-176.806,11.321,149.473
C02993=1124.910,389.137,-88.498,-176.805,11.323,149.473
C02994=1124.907,389.348,-88.531,-176.804,11.325,149.473
C02995=1124.904,389.561,-88.564,-176.803,11.327,149.474
C02996=1124.902,389.773,-88.596,-176.801,11.329,149.474
C02997=1124.898,389.986,-88.629,-176.800,11.331,149.474
C02998=1124.895,390.198,-88.662,-176.799,11.333,149.474
C02999=1124.891,390.445,-88.699,-176.797,11.335,149.474
C03000=1124.888,390.692,-88.737,-176.796,11.338,149.475
C03001=1124.884,390.939,-88.775,-176.794,11.341,149.475
C03002=1124.880,391.187,-88.812,-176.793,11.343,149.475
C03003=1124.876,391.433,-88.850,-176.792,11.345,149.476
C03004=1124.873,391.681,-88.888,-176.790,11.348,149.476
C03005=1124.869,391.927,-88.926,-176.789,11.351,149.476
C03006=1124.865,392.175,-88.964,-176.788,11.353,149.477
C03007=1124.862,392.422,-89.002,-176.787,11.355,149.477
C03008=1124.858,392.669,-89.040,-176.785,11.358,149.477
C03009=1124.854,392.916,-89.078,-176.784,11.361,149.478
C03010=1124.850,393.163,-89.116,-176.783,11.364,149.478
C03011=1124.847,393.410,-89.154,-176.782,11.366,149.478
C03012=1124.843,393.657,-89.192,-176.780,11.368,149.479
C03013=1124.839,393.904,-89.230,-176.779,11.371,149.479
C03014=1124.836,394.151,-89.268,-176.778,11.374,149.480
C03015=1124.832,394.398,-89.306,-176.777,11.377,149.480
C03016=1124.828,394.646,-89.344,-176.775,11.380,149.480
C03017=1124.825,394.892,-89.381,-176.775,11.382,149.481
C03018=1124.821,395.140,-89.420,-176.774,11.385,149.481
C03019=1124.817,395.386,-89.458,-176.772,11.388,149.482
C03020=1124.814,395.634,-89.495,-176.771,11.391,149.482
C03021=1124.810,395.881,-89.534,-176.770,11.394,149.483
C03022=1124.806,396.128,-89.572,-176.769,11.397,149.483
C03023=1124.803,396.374,-89.610,-176.768,11.400,149.484
C03024=1124.799,396.621,-89.648,-176.767,11.403,149.484
C03025=1124.795,396.868,-89.686,-176.766,11.406,149.485
C03026=1124.792,397.116,-89.725,-176.764,11.409,149.485
C03027=1124.788,397.363,-89.762,-176.763,11.412,149.486
C03028=1124.785,397.610,-89.800,-176.762,11.415,149.486
C03029=1124.781,397.858,-89.839,-176.762,11.418,149.487
C03030=1124.777,398.104,-89.876,-176.760,11.421,149.487
C03031=1124.773,398.351,-89.916,-176.759,11.424,149.488
C03032=1124.769,398.598,-89.953,-176.759,11.427,149.489
C03033=1124.766,398.845,-89.991,-176.758,11.430,149.489
C03034=1124.762,399.092,-90.030,-176.757,11.434,149.490
C03035=1124.759,399.339,-90.067,-176.756,11.437,149.490
C03036=1124.755,399.587,-90.106,-176.755,11.440,149.491
C03037=1124.752,399.833,-90.145,-176.754,11.443,149.492
C03038=1124.747,400.080,-90.183,-176.754,11.447,149.492
C03039=1124.744,400.327,-90.221,-176.753,11.450,149.493
C03040=1124.740,400.575,-90.259,-176.752,11.453,149.494
C03041=1124.737,400.821,-90.297,-176.751,11.456,149.494
C03042=1124.733,401.068,-90.335,-176.751,11.460,149.495
C03043=1124.729,401.316,-90.374,-176.750,11.463,149.496
C03044=1124.726,401.562,-90.412,-176.749,11.466,149.496
C03045=1124.722,401.809,-90.451,-176.748,11.470,149.497
C03046=1124.719,402.057,-90.489,-176.747,11.474,149.498
C03047=1124.715,402.269,-90.521,-176.747,11.476,149.498
C03048=1124.712,402.481,-90.555,-176.746,11.480,149.499
C03049=1124.709,402.693,-90.587,-176.746,11.483,149.500
C03050=1124.706,402.905,-90.620,-176.746,11.486,149.500
C03051=1124.702,403.117,-90.653,-176.745,11.489,149.501
C03052=1124.700,403.329,-90.687,-176.744,11.492,149.502
C03053=1124.696,403.542,-90.719,-176.743,11.496,149.503
C03054=1124.694,403.753,-90.752,-176.743,11.498,149.503
C03055=1124.690,404.001,-90.791,-176.742,11.503,149.504
C03056=1124.686,404.247,-90.829,-176.742,11.506,149.505
C03057=1124.682,404.494,-90.867,-176.742,11.510,149.506
C03058=1124.678,404.742,-90.906,-176.741,11.514,149.507
C03059=1124.675,404.988,-90.944,-176.740,11.518,149.507
C03060=1124.671,405.235,-90.983,-176.740,11.522,149.508
C03061=1124.668,405.482,-91.021,-176.740,11.525,149.509
C03062=1124.664,405.730,-91.060,-176.739,11.530,149.510
C03063=1124.660,405.976,-91.098,-176.739,11.534,149.511
C03064=1124.657,406.223,-91.137,-176.738,11.537,149.512
C03065=1124.654,406.470,-91.175,-176.737,11.542,149.513
C03066=1124.650,406.717,-91.214,-176.737,11.546,149.514
C03067=1124.645,406.964,-91.252,-176.737,11.549,149.515
C03068=1124.643,407.211,-91.291,-176.737,11.554,149.516
C03069=1124.639,407.459,-91.329,-176.736,11.558,149.517
C03070=1124.636,407.705,-91.368,-176.736,11.563,149.518
C03071=1124.631,407.952,-91.406,-176.736,11.567,149.519
C03072=1124.628,408.199,-91.445,-176.736,11.571,149.520
C03073=1124.624,408.446,-91.483,-176.735,11.575,149.521
C03074=1124.621,408.693,-91.523,-176.735,11.579,149.522
C03075=1124.617,408.940,-91.560,-176.734,11.584,149.523
C03076=1124.613,409.187,-91.599,-176.734,11.588,149.524
C03077=1124.609,409.434,-91.638,-176.734,11.593,149.525
C03078=1124.607,409.681,-91.677,-176.734,11.597,149.527
C03079=1124.602,409.928,-91.715,-176.734,11.602,149.528
C03080=1124.598,410.175,-91.754,-176.734,11.606,149.529
C03081=1124.596,410.422,-91.793,-176.734,11.611,149.530
C03082=1124.592,410.669,-91.831,-176.734,11.615,149.531
C03083=1124.588,410.916,-91.870,-176.734,11.620,149.532
C03084=1124.584,411.163,-91.908,-176.733,11.625,149.533
C03085=1124.581,411.410,-91.947,-176.733,11.629,149.535
C03086=1124.577,411.657,-91.987,-176.733,11.634,149.536
C03087=1124.573,411.919,-92.027,-176.733,11.639,149.537
C03088=1124.569,412.181,-92.068,-176.733,11.644,149.539
C03089=1124.566,412.443,-92.110,-176.733,11.649,149.540
C03090=1124.562,412.705,-92.151,-176.734,11.654,149.541
C03091=1124.558,412.952,-92.189,-176.733,11.659,149.543
C03092=1124.555,413.199,-92.228,-176.733,11.664,149.544
C03093=1124.551,413.446,-92.267,-176.734,11.668,149.545
C03094=1124.547,413.694,-92.306,-176.734,11.674,149.547
C03095=1124.544,413.940,-92.344,-176.734,11.679,149.548
C03096=1124.541,414.187,-92.384,-176.734,11.684,149.549
C03097=1124.539,414.433,-92.422,-176.734,11.689,149.551
C03098=1124.536,414.681,-92.461,-176.735,11.694,149.552
C03099=1124.535,414.928,-92.499,-176.735,11.700,149.553
C03100=1124.535,415.175,-92.537,-176.735,11.705,149.555
C03101=1124.535,415.422,-92.576,-176.735,11.709,149.556
C03102=1124.535,415.669,-92.614,-176.736,11.715,149.558
C03103=1124.536,416.078,-92.677,-176.736,11.723,149.560
C03104=1124.540,416.487,-92.740,-176.737,11.733,149.563
C03105=1124.545,416.895,-92.803,-176.738,11.741,149.565
C03106=1124.551,417.303,-92.866,-176.739,11.750,149.568
C03107=1124.133,417.303,-92.928,-176.731,11.755,149.567
C03108=1124.129,417.091,-92.895,-176.731,11.750,149.566
C03109=1124.126,416.880,-92.863,-176.730,11.746,149.564
C03110=1124.123,416.667,-92.831,-176.730,11.741,149.563
C03111=1124.121,416.455,-92.798,-176.730,11.736,149.562
C03112=1124.119,416.244,-92.765,-176.729,11.732,149.560
C03113=1124.117,416.032,-92.733,-176.729,11.727,149.559
C03114=1124.116,415.820,-92.700,-176.729,11.722,149.558
C03115=1124.115,415.609,-92.667,-176.728,11.718,149.557
C03116=1124.116,415.361,-92.629,-176.728,11.713,149.555
C03117=1124.115,415.114,-92.590,-176.728,11.707,149.554
C03118=1124.116,414.867,-92.552,-176.727,11.702,149.552
C03119=1124.117,414.620,-92.513,-176.727,11.697,149.551
C03120=1124.120,414.373,-92.474,-176.727,11.692,149.550
C03121=1124.122,414.126,-92.436,-176.727,11.687,149.548
C03122=1124.125,413.879,-92.397,-176.727,11.681,149.547
C03123=1124.129,413.632,-92.358,-176.727,11.676,149.546
C03124=1124.133,413.385,-92.319,-176.727,11.672,149.544
C03125=1124.136,413.138,-92.281,-176.727,11.667,149.543
C03126=1124.140,412.892,-92.242,-176.727,11.661,149.542
C03127=1124.144,412.644,-92.203,-176.727,11.656,149.540
C03128=1124.147,412.398,-92.165,-176.727,11.652,149.539
C03129=1124.150,412.151,-92.125,-176.727,11.647,149.538
C03130=1124.154,411.903,-92.087,-176.727,11.642,149.537
C03131=1124.158,411.656,-92.048,-176.727,11.638,149.535
C03132=1124.161,411.410,-92.009,-176.727,11.633,149.534
C03133=1124.165,411.163,-91.971,-176.727,11.628,149.533
C03134=1124.169,410.916,-91.932,-176.727,11.624,149.532
C03135=1124.172,410.669,-91.893,-176.727,11.619,149.530
C03136=1124.176,410.421,-91.854,-176.728,11.614,149.529
C03137=1124.180,410.175,-91.815,-176.728,11.610,149.528
C03138=1124.183,409.928,-91.777,-176.728,11.605,149.527
C03139=1124.187,409.681,-91.738,-176.729,11.600,149.526
C03140=1124.190,409.434,-91.699,-176.729,11.596,149.525
C03141=1124.194,409.187,-91.661,-176.729,11.591,149.524
C03142=1124.198,408.940,-91.622,-176.729,11.587,149.523
C03143=1124.202,408.693,-91.584,-176.730,11.582,149.522
C03144=1124.205,408.446,-91.545,-176.730,11.578,149.521
C03145=1124.208,408.199,-91.506,-176.730,11.574,149.519
C03146=1124.212,407.953,-91.468,-176.730,11.570,149.519
C03147=1124.216,407.705,-91.430,-176.731,11.565,149.517
C03148=1124.220,407.458,-91.390,-176.731,11.561,149.516
C03149=1124.223,407.211,-91.352,-176.732,11.557,149.515
C03150=1124.227,406.965,-91.314,-176.732,11.553,149.514
C03151=1124.230,406.717,-91.276,-176.732,11.549,149.514
C03152=1124.234,406.470,-91.236,-176.733,11.545,149.513
C03153=1124.238,406.223,-91.198,-176.733,11.541,149.512
C03154=1124.241,405.977,-91.160,-176.734,11.536,149.511
C03155=1124.245,405.729,-91.121,-176.734,11.533,149.510
C03156=1124.248,405.483,-91.082,-176.735,11.529,149.509
C03157=1124.252,405.235,-91.044,-176.735,11.524,149.508
C03158=1124.256,404.988,-91.006,-176.736,11.521,149.507
C03159=1124.259,404.742,-90.967,-176.736,11.517,149.506
C03160=1124.262,404.494,-90.929,-176.737,11.513,149.505
C03161=1124.266,404.247,-90.890,-176.737,11.509,149.504
C03162=1124.271,404.000,-90.852,-176.738,11.506,149.504
C03163=1124.274,403.753,-90.814,-176.739,11.501,149.503
C03164=1124.278,403.434,-90.764,-176.740,11.496,149.502
C03165=1124.283,403.114,-90.714,-176.741,11.492,149.501
C03166=1124.288,402.794,-90.665,-176.741,11.487,149.500
C03167=1124.293,402.474,-90.615,-176.743,11.482,149.499
C03168=1124.296,402.227,-90.576,-176.743,11.479,149.498
C03169=1124.300,401.979,-90.538,-176.744,11.475,149.497
C03170=1124.304,401.733,-90.499,-176.744,11.472,149.496
C03171=1124.307,401.486,-90.461,-176.745,11.468,149.496
C03172=1124.313,401.134,-90.406,-176.747,11.463,149.495
C03173=1124.318,400.783,-90.352,-176.748,11.459,149.494
C03174=1124.323,400.432,-90.298,-176.749,11.453,149.493
C03175=1124.328,400.080,-90.243,-176.750,11.449,149.492
C03176=1124.332,399.834,-90.205,-176.751,11.446,149.491
C03177=1124.335,399.586,-90.167,-176.751,11.442,149.491
C03178=1124.339,399.339,-90.129,-176.753,11.438,149.490
C03179=1124.343,399.093,-90.090,-176.754,11.435,149.489
C03180=1124.346,398.845,-90.052,-176.755,11.432,149.489
C03181=1124.351,398.599,-90.014,-176.756,11.429,149.488
C03182=1124.354,398.351,-89.976,-176.757,11.426,149.488
C03183=1124.357,398.104,-89.938,-176.757,11.422,149.487
C03184=1124.361,397.858,-89.899,-176.759,11.419,149.486
C03185=1124.364,397.610,-89.861,-176.760,11.416,149.486
C03186=1124.368,397.363,-89.823,-176.761,11.413,149.485
C03187=1124.372,397.116,-89.785,-176.762,11.410,149.485
C03188=1124.375,396.869,-89.747,-176.763,11.407,149.484
C03189=1124.380,396.622,-89.709,-176.764,11.404,149.484
C03190=1124.383,396.375,-89.671,-176.765,11.401,149.483
C03191=1124.387,396.127,-89.633,-176.766,11.398,149.483
C03192=1124.390,395.881,-89.594,-176.767,11.395,149.482
C03193=1124.394,395.634,-89.556,-176.768,11.392,149.482
C03194=1124.398,395.386,-89.518,-176.769,11.389,149.481
C03195=1124.401,395.140,-89.480,-176.771,11.387,149.481
C03196=1124.405,394.893,-89.442,-176.772,11.384,149.481
C03197=1124.409,394.646,-89.404,-176.772,11.381,149.480
C03198=1124.412,394.398,-89.366,-176.774,11.379,149.480
C03199=1124.417,394.152,-89.328,-176.775,11.376,149.479
C03200=1124.420,393.904,-89.290,-176.776,11.373,149.479
C03201=1124.423,393.657,-89.252,-176.778,11.370,149.478
C03202=1124.428,393.410,-89.214,-176.779,11.367,149.478
C03203=1124.431,393.163,-89.176,-176.781,11.365,149.478
C03204=1124.435,392.916,-89.138,-176.782,11.362,149.477
C03205=1124.439,392.669,-89.100,-176.782,11.360,149.477
C03206=1124.442,392.422,-89.062,-176.784,11.357,149.477
C03207=1124.446,392.175,-89.024,-176.785,11.354,149.476
C03208=1124.449,391.928,-88.987,-176.787,11.352,149.476
C03209=1124.453,391.681,-88.948,-176.788,11.349,149.476
C03210=1124.456,391.434,-88.910,-176.790,11.346,149.475
C03211=1124.460,391.187,-88.873,-176.791,11.344,149.475
C03212=1124.463,390.940,-88.835,-176.792,11.342,149.475
C03213=1124.468,390.692,-88.797,-176.794,11.339,149.474
C03214=1124.471,390.445,-88.759,-176.796,11.337,149.474
C03215=1124.475,390.198,-88.722,-176.796,11.335,149.474
C03216=1124.479,389.986,-88.689,-176.798,11.332,149.474
C03217=1124.482,389.774,-88.657,-176.799,11.330,149.474
C03218=1124.484,389.562,-88.624,-176.801,11.328,149.473
C03219=1124.487,389.349,-88.591,-176.802,11.326,149.473
C03220=1124.490,389.137,-88.559,-176.803,11.324,149.473
C03221=1124.494,388.925,-88.527,-176.805,11.322,149.473
C03222=1124.497,388.712,-88.494,-176.806,11.320,149.473
C03223=1124.500,388.500,-88.462,-176.807,11.318,149.472
C03224=1124.504,388.254,-88.424,-176.809,11.316,149.472
C03225=1124.508,388.006,-88.386,-176.810,11.313,149.472
C03226=1124.512,387.759,-88.349,-176.811,11.312,149.472
C03227=1124.515,387.512,-88.311,-176.813,11.309,149.472
C03228=1124.519,387.265,-88.273,-176.815,11.307,149.472
C03229=1124.523,387.018,-88.235,-176.816,11.306,149.472
C03230=1124.526,386.771,-88.197,-176.818,11.303,149.471
C03231=1124.530,386.523,-88.160,-176.820,11.300,149.471
C03232=1124.534,386.277,-88.123,-176.821,11.299,149.471
C03233=1124.537,386.029,-88.085,-176.823,11.297,149.471
C03234=1124.541,385.783,-88.047,-176.825,11.294,149.471
C03235=1124.545,385.535,-88.009,-176.826,11.293,149.471
C03236=1124.549,385.288,-87.972,-176.828,11.291,149.471
C03237=1124.552,385.041,-87.934,-176.830,11.288,149.471
C03238=1124.556,384.794,-87.897,-176.831,11.287,149.471
C03239=1124.559,384.546,-87.859,-176.833,11.284,149.470
C03240=1124.563,384.300,-87.821,-176.834,11.283,149.470
C03241=1124.567,384.053,-87.784,-176.837,11.281,149.470
C03242=1124.570,383.805,-87.747,-176.839,11.278,149.470
C03243=1124.575,383.558,-87.708,-176.840,11.277,149.470
C03244=1124.578,383.311,-87.671,-176.842,11.275,149.470
C03245=1124.582,383.064,-87.634,-176.845,11.272,149.470
C03246=1124.585,382.817,-87.596,-176.848,11.269,149.470
C03247=1124.589,382.569,-87.559,-176.851,11.267,149.470
C03248=1124.593,382.323,-87.521,-176.854,11.265,149.470
C03249=1124.597,382.075,-87.484,-176.857,11.262,149.471
C03250=1124.600,381.828,-87.446,-176.860,11.259,149.471
C03251=1124.604,381.581,-87.409,-176.862,11.257,149.471
C03252=1124.608,381.334,-87.372,-176.865,11.255,149.471
C03253=1124.611,381.086,-87.334,-176.868,11.252,149.471
C03254=1124.615,380.840,-87.297,-176.871,11.250,149.471
C03255=1124.619,380.592,-87.260,-176.874,11.247,149.471
C03256=1124.622,380.345,-87.222,-176.877,11.245,149.471
C03257=1124.626,380.098,-87.185,-176.879,11.243,149.471
C03258=1124.630,379.851,-87.148,-176.882,11.240,149.471
C03259=1124.634,379.603,-87.110,-176.885,11.238,149.472
C03260=1124.637,379.357,-87.073,-176.888,11.235,149.472
C03261=1124.641,379.110,-87.036,-176.891,11.233,149.472
C03262=1124.645,378.862,-86.998,-176.894,11.230,149.472
C03263=1124.649,378.615,-86.961,-176.897,11.228,149.472
C03264=1124.652,378.367,-86.924,-176.900,11.226,149.472
C03265=1124.656,378.121,-86.886,-176.903,11.223,149.472
C03266=1124.660,377.874,-86.849,-176.906,11.221,149.473
C03267=1124.664,377.626,-86.812,-176.909,11.218,149.473
C03268=1124.667,377.379,-86.775,-176.912,11.216,149.473
C03269=1124.672,377.132,-86.738,-176.915,11.214,149.473
C03270=1124.676,376.885,-86.701,-176.918,11.211,149.473
C03271=1124.679,376.637,-86.664,-176.921,11.209,149.473
C03272=1124.682,376.425,-86.632,-176.924,11.207,149.473
C03273=1124.685,376.213,-86.600,-176.926,11.205,149.474
C03274=1124.689,376.000,-86.568,-176.929,11.203,149.474
C03275=1124.692,375.788,-86.536,-176.931,11.201,149.474
C03276=1124.695,375.575,-86.504,-176.934,11.199,149.474
C03277=1124.698,375.363,-86.472,-176.937,11.197,149.474
C03278=1124.701,375.151,-86.441,-176.939,11.195,149.474
C03279=1124.705,374.938,-86.409,-176.942,11.193,149.474
C03280=1124.708,374.692,-86.372,-176.945,11.190,149.475
C03281=1124.712,374.444,-86.335,-176.948,11.188,149.475
C03282=1124.716,374.197,-86.299,-176.951,11.185,149.475
C03283=1124.720,373.949,-86.261,-176.954,11.183,149.475
C03284=1124.724,373.702,-86.224,-176.957,11.181,149.475
C03285=1124.727,373.456,-86.187,-176.960,11.178,149.475
C03286=1124.731,373.209,-86.151,-176.964,11.176,149.476
C03287=1124.735,372.961,-86.113,-176.967,11.173,149.476
C03288=1124.739,372.714,-86.077,-176.970,11.172,149.476
C03289=1124.742,372.467,-86.040,-176.973,11.169,149.476
C03290=1124.746,372.220,-86.003,-176.976,11.166,149.476
C03291=1124.750,371.972,-85.966,-176.979,11.164,149.477
C03292=1124.754,371.724,-85.929,-176.982,11.162,149.477
C03293=1124.757,371.478,-85.893,-176.985,11.160,149.477
C03294=1124.761,371.230,-85.856,-176.988,11.157,149.477
C03295=1124.765,370.983,-85.819,-176.992,11.155,149.477
C03296=1124.768,370.736,-85.783,-176.995,11.152,149.478
C03297=1124.772,370.488,-85.746,-176.998,11.150,149.478
C03298=1124.776,370.241,-85.710,-177.001,11.148,149.478
C03299=1124.780,369.994,-85.673,-177.004,11.146,149.478
C03300=1124.784,369.747,-85.637,-177.008,11.143,149.479
C03301=1124.788,369.499,-85.600,-177.011,11.141,149.479
C03302=1124.791,369.252,-85.563,-177.014,11.138,149.479
C03303=1124.795,369.005,-85.526,-177.017,11.136,149.479
C03304=1124.799,368.757,-85.489,-177.020,11.134,149.479
C03305=1124.803,368.510,-85.454,-177.023,11.132,149.480
C03306=1124.807,368.263,-85.417,-177.027,11.129,149.480
C03307=1124.810,368.016,-85.381,-177.030,11.127,149.480
C03308=1124.814,367.769,-85.344,-177.034,11.125,149.480
C03309=1124.818,367.521,-85.307,-177.037,11.122,149.481
C03310=1124.821,367.273,-85.271,-177.040,11.120,149.481
C03311=1124.825,367.026,-85.234,-177.043,11.118,149.481
C03312=1124.829,366.779,-85.198,-177.046,11.115,149.481
C03313=1124.833,366.531,-85.162,-177.050,11.113,149.482
C03314=1124.837,366.284,-85.126,-177.053,11.111,149.482
C03315=1124.841,366.037,-85.089,-177.056,11.108,149.482
C03316=1124.845,365.789,-85.053,-177.060,11.106,149.482
C03317=1124.848,365.543,-85.016,-177.063,11.103,149.483
C03318=1124.852,365.295,-84.979,-177.066,11.101,149.483
C03319=1124.856,365.048,-84.944,-177.070,11.098,149.483
C03320=1124.860,364.801,-84.907,-177.072,11.097,149.483
C03321=1124.864,364.553,-84.871,-177.076,11.094,149.483
C03322=1124.867,364.306,-84.835,-177.079,11.092,149.484
C03323=1124.871,364.058,-84.798,-177.083,11.090,149.484
C03324=1124.874,363.811,-84.762,-177.086,11.087,149.484
C03325=1124.878,363.564,-84.726,-177.089,11.085,149.484
C03326=1124.882,363.316,-84.690,-177.093,11.082,149.485
C03327=1124.886,363.069,-84.653,-177.096,11.080,149.485
C03328=1124.890,362.857,-84.622,-177.099,11.078,149.485
C03329=1124.893,362.644,-84.592,-177.102,11.076,149.485
C03330=1124.896,362.431,-84.561,-177.105,11.074,149.486
C03331=1124.899,362.220,-84.530,-177.108,11.071,149.486
C03332=1124.902,362.007,-84.499,-177.111,11.070,149.486
C03333=1124.905,361.794,-84.468,-177.113,11.068,149.486
C03334=1124.909,361.582,-84.437,-177.117,11.066,149.487
C03335=1124.912,361.369,-84.406,-177.119,11.064,149.487
C03336=1124.916,361.122,-84.370,-177.123,11.061,149.487
C03337=1124.920,360.874,-84.334,-177.126,11.059,149.487
C03338=1124.924,360.627,-84.298,-177.129,11.057,149.487
C03339=1124.927,360.380,-84.262,-177.133,11.054,149.488
C03340=1124.931,360.132,-84.226,-177.136,11.052,149.488
C03341=1124.935,359.885,-84.190,-177.140,11.049,149.488
C03342=1124.938,359.638,-84.154,-177.143,11.047,149.489
C03343=1124.943,359.390,-84.118,-177.147,11.045,149.489
C03344=1124.947,359.142,-84.082,-177.150,11.042,149.489
C03345=1124.950,358.896,-84.046,-177.154,11.039,149.489
C03346=1124.954,358.648,-84.010,-177.157,11.037,149.490
C03347=1124.959,358.401,-83.975,-177.161,11.035,149.490
C03348=1124.962,358.153,-83.939,-177.164,11.032,149.490
C03349=1124.966,357.906,-83.904,-177.167,11.030,149.490
C03350=1124.970,357.658,-83.868,-177.171,11.027,149.491
C03351=1124.974,357.411,-83.831,-177.174,11.025,149.491
C03352=1124.977,357.164,-83.796,-177.178,11.023,149.491
C03353=1124.981,356.916,-83.760,-177.181,11.020,149.491
C03354=1124.985,356.669,-83.725,-177.184,11.018,149.492
C03355=1124.988,356.421,-83.689,-177.188,11.015,149.492
C03356=1124.993,356.174,-83.654,-177.192,11.012,149.492
C03357=1124.997,355.927,-83.618,-177.195,11.010,149.492
C03358=1125.001,355.679,-83.582,-177.199,11.007,149.493
C03359=1125.004,355.432,-83.547,-177.202,11.005,149.493
C03360=1125.008,355.184,-83.511,-177.206,11.003,149.493
C03361=1125.012,354.937,-83.475,-177.209,11.000,149.494
C03362=1125.015,354.689,-83.440,-177.212,10.998,149.494
C03363=1125.020,354.442,-83.405,-177.216,10.995,149.494
C03364=1125.023,354.195,-83.369,-177.220,10.992,149.494
C03365=1125.028,353.947,-83.333,-177.223,10.990,149.495
C03366=1125.031,353.700,-83.297,-177.226,10.987,149.495
C03367=1125.035,353.452,-83.262,-177.230,10.985,149.495
C03368=1125.039,353.205,-83.227,-177.234,10.982,149.495
C03369=1125.043,352.958,-83.191,-177.237,10.980,149.496
C03370=1125.047,352.710,-83.156,-177.241,10.977,149.496
C03371=1125.050,352.462,-83.121,-177.244,10.975,149.496
C03372=1125.054,352.215,-83.085,-177.248,10.971,149.496
C03373=1125.058,351.968,-83.050,-177.252,10.969,149.497
C03374=1125.062,351.720,-83.015,-177.255,10.967,149.497
C03375=1125.066,351.473,-82.979,-177.258,10.964,149.497
C03376=1125.070,351.225,-82.944,-177.262,10.961,149.497
C03377=1125.074,350.978,-82.909,-177.266,10.959,149.498
C03378=1125.078,350.730,-82.873,-177.269,10.957,149.498
C03379=1125.081,350.483,-82.838,-177.273,10.954,149.498
C03380=1125.085,350.235,-82.803,-177.277,10.951,149.498
C03381=1125.090,349.988,-82.768,-177.280,10.948,149.499
C03382=1125.093,349.740,-82.732,-177.283,10.946,149.499
C03383=1125.097,349.492,-82.697,-177.287,10.943,149.499
C03384=1125.100,349.280,-82.668,-177.290,10.941,149.499
C03385=1125.104,349.068,-82.638,-177.293,10.939,149.500
C03386=1125.107,348.855,-82.607,-177.295,10.937,149.500
C03387=1125.111,348.643,-82.577,-177.298,10.935,149.500
C03388=1125.113,348.430,-82.547,-177.301,10.932,149.500
C03389=1125.117,348.217,-82.517,-177.304,10.930,149.500
C03390=1125.120,348.005,-82.487,-177.306,10.929,149.500
C03391=1125.124,347.792,-82.457,-177.309,10.926,149.500
C03392=1125.128,347.544,-82.422,-177.313,10.923,149.501
C03393=1125.132,347.297,-82.386,-177.316,10.921,149.501
C03394=1125.136,347.049,-82.352,-177.319,10.919,149.501
C03395=1125.139,346.802,-82.317,-177.323,10.916,149.501
C03396=1125.143,346.554,-82.282,-177.326,10.914,149.502
C03397=1125.147,346.306,-82.247,-177.329,10.911,149.502
C03398=1125.152,346.059,-82.212,-177.332,10.908,149.502
C03399=1125.155,345.811,-82.177,-177.335,10.907,149.502
C03400=1125.159,345.564,-82.142,-177.338,10.904,149.502
C03401=1125.163,345.317,-82.107,-177.341,10.902,149.503
C03402=1125.167,345.069,-82.072,-177.345,10.899,149.503
C03403=1125.171,344.821,-82.038,-177.348,10.897,149.503
C03404=1125.174,344.574,-82.003,-177.351,10.894,149.503
C03405=1125.178,344.326,-81.968,-177.354,10.892,149.503
C03406=1125.183,344.079,-81.934,-177.358,10.889,149.504
C03407=1125.186,343.831,-81.898,-177.361,10.887,149.504
C03408=1125.190,343.584,-81.864,-177.364,10.884,149.504
C03409=1125.194,343.336,-81.829,-177.367,10.882,149.504
C03410=1125.199,343.089,-81.794,-177.370,10.879,149.504
C03411=1125.202,342.841,-81.759,-177.374,10.877,149.505
C03412=1125.206,342.594,-81.726,-177.377,10.874,149.505
C03413=1125.210,342.346,-81.691,-177.380,10.872,149.505
C03414=1125.214,342.098,-81.656,-177.384,10.869,149.505
C03415=1125.218,341.851,-81.621,-177.387,10.866,149.505
C03416=1125.222,341.603,-81.586,-177.390,10.864,149.506
C03417=1125.226,341.356,-81.552,-177.393,10.862,149.506
C03418=1125.230,341.108,-81.518,-177.397,10.859,149.506
C03419=1125.234,340.860,-81.483,-177.399,10.857,149.506
C03420=1125.237,340.613,-81.449,-177.403,10.855,149.507
C03421=1125.242,340.366,-81.414,-177.405,10.852,149.507
C03422=1125.246,340.118,-81.379,-177.409,10.850,149.507
C03423=1125.249,339.871,-81.345,-177.412,10.847,149.507
C03424=1125.253,339.622,-81.310,-177.415,10.845,149.507
C03425=1125.257,339.375,-81.276,-177.418,10.842,149.507
C03426=1125.262,339.128,-81.242,-177.422,10.840,149.508
C03427=1125.266,338.880,-81.207,-177.425,10.837,149.508
C03428=1125.270,338.633,-81.173,-177.428,10.835,149.508
C03429=1125.274,338.385,-81.138,-177.432,10.832,149.508
C03430=1125.277,338.137,-81.105,-177.434,10.829,149.508
C03431=1125.281,337.889,-81.070,-177.438,10.827,149.509
C03432=1125.285,337.642,-81.036,-177.441,10.824,149.509
C03433=1125.289,337.394,-81.001,-177.444,10.822,149.509
C03434=1125.293,337.147,-80.967,-177.448,10.820,149.509
C03435=1125.298,336.900,-80.933,-177.451,10.817,149.509
C03436=1125.301,336.651,-80.899,-177.454,10.814,149.510
C03437=1125.306,336.404,-80.865,-177.457,10.812,149.510
C03438=1125.309,336.156,-80.831,-177.460,10.810,149.510
C03439=1125.313,335.909,-80.797,-177.463,10.807,149.510
C03440=1125.317,335.696,-80.766,-177.466,10.805,149.510
C03441=1125.320,335.483,-80.737,-177.469,10.803,149.510
C03442=1125.323,335.270,-80.708,-177.472,10.801,149.511
C03443=1125.326,335.057,-80.679,-177.474,10.799,149.511
C03444=1125.330,334.845,-80.650,-177.477,10.797,149.511
C03445=1125.333,334.632,-80.620,-177.480,10.794,149.511
C03446=1125.337,334.419,-80.591,-177.482,10.792,149.511
C03447=1125.340,334.206,-80.562,-177.485,10.790,149.511
C03448=1125.344,333.958,-80.528,-177.488,10.788,149.512
C03449=1125.348,333.711,-80.494,-177.491,10.786,149.512
C03450=1125.352,333.463,-80.460,-177.495,10.783,149.512
C03451=1125.356,333.215,-80.426,-177.498,10.780,149.512
C03452=1125.360,332.968,-80.392,-177.501,10.778,149.512
C03453=1125.364,332.720,-80.358,-177.504,10.775,149.513
C03454=1125.368,332.473,-80.324,-177.508,10.773,149.513
C03455=1125.372,332.225,-80.290,-177.510,10.770,149.513
C03456=1125.375,331.977,-80.257,-177.514,10.768,149.513
C03457=1125.380,331.730,-80.222,-177.517,10.765,149.513
C03458=1125.384,331.482,-80.188,-177.520,10.763,149.514
C03459=1125.387,331.234,-80.155,-177.523,10.760,149.514
C03460=1125.392,330.987,-80.120,-177.527,10.758,149.514
C03461=1125.396,330.739,-80.087,-177.530,10.755,149.514
C03462=1125.400,330.492,-80.053,-177.533,10.752,149.514
C03463=1125.403,330.243,-80.020,-177.536,10.750,149.515
C03464=1125.408,329.996,-79.985,-177.540,10.747,149.515
C03465=1125.412,329.748,-79.952,-177.543,10.745,149.515
C03466=1125.415,329.500,-79.918,-177.545,10.743,149.515
C03467=1125.419,329.253,-79.885,-177.548,10.741,149.515
C03468=1125.423,329.006,-79.851,-177.552,10.738,149.516
C03469=1125.428,328.757,-79.817,-177.555,10.735,149.516
C03470=1125.431,328.510,-79.783,-177.558,10.733,149.516
C03471=1125.436,328.262,-79.750,-177.561,10.730,149.516
C03472=1125.440,328.014,-79.716,-177.565,10.728,149.516
C03473=1125.443,327.767,-79.683,-177.568,10.725,149.516
C03474=1125.448,327.519,-79.649,-177.571,10.723,149.517
C03475=1125.451,327.272,-79.615,-177.574,10.720,149.517
C03476=1125.456,327.024,-79.581,-177.577,10.718,149.517
C03477=1125.460,326.776,-79.548,-177.581,10.715,149.517
C03478=1125.464,326.529,-79.514,-177.584,10.713,149.518
C03479=1125.467,326.280,-79.481,-177.587,10.710,149.518
C03480=1125.471,326.033,-79.448,-177.590,10.707,149.518
C03481=1125.476,325.785,-79.415,-177.593,10.705,149.518
C03482=1125.479,325.538,-79.381,-177.596,10.702,149.518
C03483=1125.483,325.290,-79.348,-177.599,10.701,149.518
C03484=1125.488,325.042,-79.314,-177.602,10.698,149.519
C03485=1125.491,324.794,-79.281,-177.605,10.695,149.519
C03486=1125.495,324.547,-79.247,-177.609,10.693,149.519
C03487=1125.499,324.299,-79.214,-177.612,10.690,149.519
C03488=1125.503,324.051,-79.181,-177.615,10.688,149.519
C03489=1125.507,323.804,-79.148,-177.618,10.685,149.520
C03490=1125.512,323.556,-79.114,-177.621,10.683,149.520
C03491=1125.515,323.307,-79.081,-177.624,10.680,149.520
C03492=1125.519,323.060,-79.048,-177.628,10.678,149.520
C03493=1125.523,322.813,-79.014,-177.631,10.675,149.520
C03494=1125.527,322.565,-78.981,-177.634,10.672,149.520
C03495=1125.531,322.317,-78.948,-177.637,10.670,149.521
C03496=1125.535,322.104,-78.919,-177.640,10.668,149.521
C03497=1125.539,321.891,-78.890,-177.643,10.665,149.521
C03498=1125.541,321.678,-78.862,-177.645,10.663,149.521
C03499=1125.545,321.465,-78.833,-177.648,10.662,149.521
C03500=1125.549,321.252,-78.805,-177.651,10.659,149.521
C03501=1125.552,321.039,-78.777,-177.654,10.657,149.522
C03502=1125.555,320.826,-78.748,-177.656,10.655,149.522
C03503=1125.559,320.613,-78.720,-177.659,10.653,149.522
C03504=1125.563,320.365,-78.687,-177.662,10.650,149.522
C03505=1125.567,320.117,-78.653,-177.665,10.648,149.522
C03506=1125.571,319.870,-78.621,-177.668,10.645,149.522
C03507=1125.575,319.622,-78.588,-177.672,10.642,149.523
C03508=1125.579,319.374,-78.555,-177.675,10.640,149.523
C03509=1125.583,319.127,-78.521,-177.677,10.638,149.523
C03510=1125.587,318.879,-78.488,-177.681,10.636,149.523
C03511=1125.591,318.632,-78.456,-177.684,10.633,149.524
C03512=1125.595,318.383,-78.423,-177.687,10.630,149.524
C03513=1125.599,318.135,-78.390,-177.690,10.628,149.524
C03514=1125.603,317.888,-78.357,-177.693,10.625,149.524
C03515=1125.607,317.640,-78.324,-177.696,10.623,149.524
C03516=1125.611,317.393,-78.291,-177.700,10.620,149.524
C03517=1125.615,317.144,-78.259,-177.703,10.617,149.525
C03518=1125.619,316.897,-78.226,-177.706,10.615,149.525
C03519=1125.624,316.649,-78.193,-177.709,10.613,149.525
C03520=1125.627,316.401,-78.160,-177.712,10.610,149.525
C03521=1125.631,316.153,-78.128,-177.716,10.607,149.525
C03522=1125.636,315.905,-78.094,-177.719,10.605,149.525
C03523=1125.640,315.658,-78.061,-177.722,10.602,149.526
C03524=1125.643,315.410,-78.029,-177.725,10.601,149.526
C03525=1125.647,315.162,-77.996,-177.727,10.598,149.526
C03526=1125.652,314.914,-77.963,-177.731,10.595,149.526
C03527=1125.655,314.666,-77.931,-177.734,10.593,149.526
C03528=1125.659,314.418,-77.898,-177.737,10.590,149.527
C03529=1125.664,314.171,-77.865,-177.740,10.588,149.527
C03530=1125.667,313.923,-77.833,-177.743,10.585,149.527
C03531=1125.671,313.675,-77.800,-177.747,10.582,149.527
C03532=1125.676,313.426,-77.767,-177.750,10.580,149.527
C03533=1125.679,313.179,-77.735,-177.753,10.577,149.528
C03534=1125.684,312.931,-77.702,-177.756,10.575,149.528
C03535=1125.688,312.684,-77.670,-177.759,10.572,149.528
C03536=1125.692,312.436,-77.638,-177.762,10.570,149.528
C03537=1125.696,312.188,-77.605,-177.765,10.567,149.528
C03538=1125.700,311.940,-77.573,-177.769,10.564,149.528
C03539=1125.704,311.692,-77.540,-177.771,10.563,149.529
C03540=1125.708,311.444,-77.508,-177.774,10.560,149.529
C03541=1125.712,311.196,-77.475,-177.778,10.558,149.529
C03542=1125.716,310.948,-77.443,-177.781,10.555,149.529
C03543=1125.720,310.701,-77.410,-177.784,10.552,149.529
C03544=1125.724,310.453,-77.378,-177.787,10.550,149.529
C03545=1125.729,310.205,-77.346,-177.790,10.547,149.530
C03546=1125.732,309.957,-77.313,-177.794,10.545,149.530
C03547=1125.736,309.709,-77.281,-177.796,10.542,149.530
C03548=1125.740,309.461,-77.249,-177.800,10.539,149.530
C03549=1125.745,309.214,-77.216,-177.803,10.537,149.530
C03550=1125.749,308.966,-77.184,-177.806,10.534,149.531
C03551=1125.753,308.718,-77.152,-177.809,10.531,149.531
C03552=1125.756,308.504,-77.124,-177.812,10.530,149.531
C03553=1125.760,308.291,-77.096,-177.814,10.528,149.531
C03554=1125.764,308.078,-77.069,-177.817,10.525,149.531
C03555=1125.767,307.865,-77.041,-177.820,10.523,149.532
C03556=1125.771,307.652,-77.013,-177.822,10.521,149.532
C03557=1125.774,307.439,-76.986,-177.825,10.519,149.532
C03558=1125.777,307.226,-76.958,-177.828,10.517,149.532
C03559=1125.781,307.013,-76.930,-177.830,10.514,149.532
C03560=1125.785,306.765,-76.898,-177.834,10.512,149.532
C03561=1125.789,306.518,-76.866,-177.836,10.510,149.532
C03562=1125.793,306.270,-76.834,-177.839,10.507,149.533
C03563=1125.797,306.021,-76.802,-177.842,10.505,149.533
C03564=1125.801,305.773,-76.769,-177.846,10.502,149.533
C03565=1125.806,305.526,-76.738,-177.849,10.499,149.533
C03566=1125.810,305.278,-76.706,-177.852,10.497,149.533
C03567=1125.814,305.029,-76.674,-177.855,10.495,149.534
C03568=1125.818,304.781,-76.642,-177.858,10.492,149.534
C03569=1125.822,304.534,-76.610,-177.862,10.489,149.534
C03570=1125.826,304.286,-76.578,-177.864,10.487,149.534
C03571=1125.830,304.038,-76.546,-177.868,10.484,149.534
C03572=1125.834,303.790,-76.515,-177.871,10.481,149.534
C03573=1125.839,303.542,-76.482,-177.874,10.479,149.535
C03574=1125.843,303.294,-76.450,-177.876,10.477,149.535
C03575=1125.847,303.047,-76.419,-177.880,10.474,149.535
C03576=1125.851,302.799,-76.387,-177.883,10.472,149.535
C03577=1125.855,302.550,-76.354,-177.886,10.469,149.535
C03578=1125.859,302.303,-76.323,-177.889,10.467,149.535
C03579=1125.863,302.055,-76.291,-177.892,10.464,149.536
C03580=1125.867,301.807,-76.259,-177.895,10.461,149.536
C03581=1125.872,301.559,-76.227,-177.899,10.459,149.536
C03582=1125.875,301.311,-76.195,-177.901,10.456,149.536
C03583=1125.879,301.063,-76.164,-177.905,10.454,149.536
C03584=1125.884,300.815,-76.133,-177.908,10.451,149.536
C03585=1125.888,300.567,-76.100,-177.911,10.448,149.537
C03586=1125.892,300.319,-76.069,-177.914,10.447,149.537
C03587=1125.896,300.071,-76.037,-177.917,10.444,149.537
C03588=1125.900,299.823,-76.005,-177.920,10.442,149.537
C03589=1125.905,299.575,-75.974,-177.923,10.439,149.537
C03590=1125.908,299.327,-75.943,-177.926,10.436,149.538
C03591=1125.912,299.079,-75.911,-177.929,10.434,149.538
C03592=1125.917,298.832,-75.879,-177.933,10.431,149.538
C03593=1125.921,298.583,-75.848,-177.935,10.428,149.538
C03594=1125.925,298.336,-75.816,-177.939,10.426,149.538
C03595=1125.929,298.088,-75.784,-177.942,10.423,149.539
C03596=1125.933,297.839,-75.753,-177.945,10.421,149.539
C03597=1125.937,297.592,-75.722,-177.948,10.418,149.539
C03598=1125.941,297.344,-75.690,-177.951,10.416,149.539
C03599=1125.946,297.096,-75.659,-177.954,10.414,149.539
C03600=1125.949,296.848,-75.627,-177.957,10.411,149.540
C03601=1125.954,296.600,-75.596,-177.960,10.408,149.540
C03602=1125.958,296.352,-75.565,-177.963,10.406,149.540
C03603=1125.962,296.104,-75.533,-177.966,10.403,149.540
C03604=1125.966,295.856,-75.502,-177.970,10.401,149.540
C03605=1125.970,295.608,-75.470,-177.972,10.398,149.540
C03606=1125.974,295.360,-75.439,-177.975,10.395,149.540
C03607=1125.978,295.112,-75.407,-177.979,10.393,149.541
C03608=1125.982,294.898,-75.381,-177.981,10.391,149.541
C03609=1125.985,294.685,-75.353,-177.984,10.389,149.541
C03610=1125.989,294.472,-75.327,-177.987,10.387,149.541
C03611=1125.993,294.258,-75.300,-177.989,10.385,149.541
C03612=1125.996,294.046,-75.273,-177.992,10.382,149.541
C03613=1126.000,293.832,-75.246,-177.995,10.380,149.542
C03614=1126.004,293.619,-75.219,-177.997,10.378,149.542
C03615=1126.007,293.405,-75.193,-178.000,10.375,149.542
C03616=1126.011,293.158,-75.161,-178.003,10.373,149.542
C03617=1126.015,292.909,-75.131,-178.006,10.371,149.542
C03618=1126.019,292.662,-75.099,-178.009,10.369,149.543
C03619=1126.023,292.413,-75.068,-178.012,10.366,149.543
C03620=1126.028,292.165,-75.037,-178.015,10.363,149.543
C03621=1126.031,291.917,-75.005,-178.018,10.361,149.543
C03622=1126.036,291.669,-74.975,-178.021,10.358,149.543
C03623=1126.040,291.421,-74.944,-178.024,10.355,149.543
C03624=1126.043,291.174,-74.913,-178.027,10.353,149.543
C03625=1126.048,290.926,-74.882,-178.031,10.350,149.544
C03626=1126.052,290.677,-74.851,-178.034,10.347,149.544
C03627=1126.057,290.429,-74.820,-178.037,10.345,149.544
C03628=1126.060,290.181,-74.788,-178.039,10.343,149.544
C03629=1126.065,289.933,-74.757,-178.043,10.341,149.544
C03630=1126.069,289.686,-74.727,-178.045,10.338,149.545
C03631=1126.073,289.437,-74.696,-178.049,10.335,149.545
C03632=1126.077,289.190,-74.665,-178.052,10.333,149.545
C03633=1126.081,288.941,-74.633,-178.055,10.330,149.545
C03634=1126.085,288.693,-74.603,-178.058,10.327,149.545
C03635=1126.090,288.445,-74.573,-178.061,10.325,149.545
C03636=1126.094,288.197,-74.541,-178.064,10.322,149.546
C03637=1126.098,287.949,-74.511,-178.067,10.320,149.546
C03638=1126.102,287.701,-74.480,-178.070,10.318,149.546
C03639=1126.106,287.452,-74.449,-178.073,10.315,149.546
C03640=1126.111,287.205,-74.418,-178.076,10.313,149.546
C03641=1126.114,286.957,-74.388,-178.079,10.310,149.547
C03642=1126.118,286.709,-74.357,-178.082,10.307,149.547
C03643=1126.123,286.461,-74.326,-178.085,10.305,149.547
C03644=1126.127,286.213,-74.296,-178.088,10.302,149.547
C03645=1126.131,285.964,-74.264,-178.092,10.300,149.547
C03646=1126.136,285.716,-74.234,-178.095,10.297,149.547
C03647=1126.139,285.469,-74.204,-178.098,10.294,149.548
